FUNCTION_BLOCK "DEVTYPE_ODH_Area"
{ S7_Optimized_Access := 'TRUE' }
VERSION : 1.0
   VAR_INPUT
      "Alarm" { S7_HMI_Accessible := 'False'; S7_HMI_Visible := 'False'} : BOOL;   //EPICS Status variable: Alarm
      "WarmUp" { S7_HMI_Accessible := 'False'; S7_HMI_Visible := 'False'} : BOOL;   //EPICS Status variable: WarmUp
      "ConnLost" { S7_HMI_Accessible := 'False'; S7_HMI_Visible := 'False'} : BOOL;   //EPICS Status variable: ConnLost
   END_VAR
   VAR_OUTPUT
      DEVICE_PARAM_OK { S7_HMI_Accessible := 'False'; S7_HMI_Visible := 'False'} : Bool;
   END_VAR
   VAR_IN_OUT
   END_VAR
   VAR
      StatusReg { S7_HMI_Accessible := 'False'; S7_HMI_Visible := 'False'} : Array[0..0] of Word;
      CommandReg { S7_HMI_Accessible := 'False'; S7_HMI_Visible := 'False'} : Array[0..0] of Word;
   END_VAR
   Var DB_SPECIFIC
      MyWord { S7_HMI_Accessible := 'False'; S7_HMI_Visible := 'False'} : Word;
      MyBytesinWord { S7_HMI_Accessible := 'False'; S7_HMI_Visible := 'False'} AT MyWord : Array[0..1] of Byte;
      MyBoolsinWord { S7_HMI_Accessible := 'False'; S7_HMI_Visible := 'False'} AT MyWord : Array[0..15] of Bool;
      MyDInt { S7_HMI_Accessible := 'False'; S7_HMI_Visible := 'False'} : DInt;
      MyWordsinDint { S7_HMI_Accessible := 'False'; S7_HMI_Visible := 'False'} AT MyDInt : Array[0..1] of Word;
      MyReal { S7_HMI_Accessible := 'False'; S7_HMI_Visible := 'False'} : Real;
      MyWordsinReal { S7_HMI_Accessible := 'False'; S7_HMI_Visible := 'False'} AT MyReal : Array[0..1] of Word;
      MyInt { S7_HMI_Accessible := 'False'; S7_HMI_Visible := 'False'} : Int;
      MyWordinInt { S7_HMI_Accessible := 'False'; S7_HMI_Visible := 'False'} AT MyInt : Word;
      MyDWord { S7_HMI_Accessible := 'False'; S7_HMI_Visible := 'False'} : DWord;
      MyWordsinDWord { S7_HMI_Accessible := 'False'; S7_HMI_Visible := 'False'} AT MyDWord : Array[0..1] of Word;
      MyTime { S7_HMI_Accessible := 'False'; S7_HMI_Visible := 'False'} : Time;
      MyWordsinTime { S7_HMI_Accessible := 'False'; S7_HMI_Visible := 'False'} AT MyTime : Array[0..1] of Word;
   END_VAR
   VAR_TEMP
      HashModbus : DInt;
      HashIFA : DInt;
      HashTIAMap : DInt;
   END_VAR
    //Author: Miklos Boros (miklos.boros@esss.se), Copyrigth 2017-2018 by European Spallation Source, Lund
    //This block was generated by PLCFactory, please don't change it MANUALLY!
    //Input File Name: KG-GTA_ODH-PLC-01-template-IFA-20181024185957.ifa
    //According to HASH: 733470530
    //Device type: ODH_Area
    //Generated: 20181024185959
    //Description: This function does the variable mapping for a device. All device-variable will be linked to an interface variable defined in this block.

    //********************************************
    //****************HASH check******************
    //********************************************


    #MyWordsinDint[0] := "EPICSToPLC"."Word"[0];
    #MyWordsinDint[1] := "EPICSToPLC"."Word"[1];
    #HashModbus := #MyDInt; //Hash from EPICS/ModbusTCP

    #HashIFA := 733470530; //Hash from Interface Factory as a constant

    #MyWordsinDint[0] := "PLCToEPICS"."Word"[0];
    #MyWordsinDint[1] := "PLCToEPICS"."Word"[1];
    #HashTIAMap := #MyDInt; //Hash from PLCFactory TIA Map


    IF ((#HashIFA = #HashModbus) AND (#HashModbus = #HashTIAMap)) THEN //Check CRCs
        #DEVICE_PARAM_OK := TRUE;
       //########################### ODH Detection System   ##############################
       //###########################
       //STATUS BLOCK
       //###########################

    //********************************************
    //*************STATUS VARIABLES***************
    //********************************************


       #MyWord := W#0;
       #MyBoolsinWord[8] := #"Alarm";    //EPICSName: Alarm
       #MyBoolsinWord[9] := #"WarmUp";    //EPICSName: WarmUp
       #MyBoolsinWord[10] := #"ConnLost";    //EPICSName: ConnLost
       #StatusReg[0] := #MyWord;
    Else
       #DEVICE_PARAM_OK := FALSE; //Invalid Hash
    END_IF;
END_FUNCTION_BLOCK
FUNCTION_BLOCK "DEVTYPE_ODH_O2iM"
{ S7_Optimized_Access := 'TRUE' }
VERSION : 1.0
   VAR_INPUT
      "O2Level" { S7_HMI_Accessible := 'False'; S7_HMI_Visible := 'False'} : REAL;   //EPICS Status variable: O2Level
      "ODHAlarm" { S7_HMI_Accessible := 'False'; S7_HMI_Visible := 'False'} : BOOL;   //EPICS Status variable: ODHAlarm
      "ODHWarning" { S7_HMI_Accessible := 'False'; S7_HMI_Visible := 'False'} : BOOL;   //EPICS Status variable: ODHWarning
      "MonitHealthy" { S7_HMI_Accessible := 'False'; S7_HMI_Visible := 'False'} : BOOL;   //EPICS Status variable: MonitHealthy
      "Maint" { S7_HMI_Accessible := 'False'; S7_HMI_Visible := 'False'} : BOOL;   //EPICS Status variable: Maint
      "MonitWarning" { S7_HMI_Accessible := 'False'; S7_HMI_Visible := 'False'} : BOOL;   //EPICS Status variable: MonitWarning
      "SysOK" { S7_HMI_Accessible := 'False'; S7_HMI_Visible := 'False'} : BOOL;   //EPICS Status variable: SysOK
      "WarmUp" { S7_HMI_Accessible := 'False'; S7_HMI_Visible := 'False'} : BOOL;   //EPICS Status variable: WarmUp
      "ConnLost" { S7_HMI_Accessible := 'False'; S7_HMI_Visible := 'False'} : BOOL;   //EPICS Status variable: ConnLost
   END_VAR
   VAR_OUTPUT
      DEVICE_PARAM_OK { S7_HMI_Accessible := 'False'; S7_HMI_Visible := 'False'} : Bool;
   END_VAR
   VAR_IN_OUT
   END_VAR
   VAR
      StatusReg { S7_HMI_Accessible := 'False'; S7_HMI_Visible := 'False'} : Array[0..2] of Word;
      CommandReg { S7_HMI_Accessible := 'False'; S7_HMI_Visible := 'False'} : Array[0..0] of Word;
   END_VAR
   Var DB_SPECIFIC
      MyWord { S7_HMI_Accessible := 'False'; S7_HMI_Visible := 'False'} : Word;
      MyBytesinWord { S7_HMI_Accessible := 'False'; S7_HMI_Visible := 'False'} AT MyWord : Array[0..1] of Byte;
      MyBoolsinWord { S7_HMI_Accessible := 'False'; S7_HMI_Visible := 'False'} AT MyWord : Array[0..15] of Bool;
      MyDInt { S7_HMI_Accessible := 'False'; S7_HMI_Visible := 'False'} : DInt;
      MyWordsinDint { S7_HMI_Accessible := 'False'; S7_HMI_Visible := 'False'} AT MyDInt : Array[0..1] of Word;
      MyReal { S7_HMI_Accessible := 'False'; S7_HMI_Visible := 'False'} : Real;
      MyWordsinReal { S7_HMI_Accessible := 'False'; S7_HMI_Visible := 'False'} AT MyReal : Array[0..1] of Word;
      MyInt { S7_HMI_Accessible := 'False'; S7_HMI_Visible := 'False'} : Int;
      MyWordinInt { S7_HMI_Accessible := 'False'; S7_HMI_Visible := 'False'} AT MyInt : Word;
      MyDWord { S7_HMI_Accessible := 'False'; S7_HMI_Visible := 'False'} : DWord;
      MyWordsinDWord { S7_HMI_Accessible := 'False'; S7_HMI_Visible := 'False'} AT MyDWord : Array[0..1] of Word;
      MyTime { S7_HMI_Accessible := 'False'; S7_HMI_Visible := 'False'} : Time;
      MyWordsinTime { S7_HMI_Accessible := 'False'; S7_HMI_Visible := 'False'} AT MyTime : Array[0..1] of Word;
   END_VAR
   VAR_TEMP
      HashModbus : DInt;
      HashIFA : DInt;
      HashTIAMap : DInt;
   END_VAR
    //Author: Miklos Boros (miklos.boros@esss.se), Copyrigth 2017-2018 by European Spallation Source, Lund
    //This block was generated by PLCFactory, please don't change it MANUALLY!
    //Input File Name: KG-GTA_ODH-PLC-01-template-IFA-20181024185957.ifa
    //According to HASH: 733470530
    //Device type: ODH_O2iM
    //Generated: 20181024185959
    //Description: This function does the variable mapping for a device. All device-variable will be linked to an interface variable defined in this block.

    //********************************************
    //****************HASH check******************
    //********************************************


    #MyWordsinDint[0] := "EPICSToPLC"."Word"[0];
    #MyWordsinDint[1] := "EPICSToPLC"."Word"[1];
    #HashModbus := #MyDInt; //Hash from EPICS/ModbusTCP

    #HashIFA := 733470530; //Hash from Interface Factory as a constant

    #MyWordsinDint[0] := "PLCToEPICS"."Word"[0];
    #MyWordsinDint[1] := "PLCToEPICS"."Word"[1];
    #HashTIAMap := #MyDInt; //Hash from PLCFactory TIA Map


    IF ((#HashIFA = #HashModbus) AND (#HashModbus = #HashTIAMap)) THEN //Check CRCs
        #DEVICE_PARAM_OK := TRUE;
       //########################### ODH Detection System   ##############################
       //###########################
       //STATUS BLOCK
       //###########################

    //********************************************
    //*************STATUS VARIABLES***************
    //********************************************


       #MyReal := #"O2Level";
       #StatusReg[0] := #MyWordsinReal[0];
       #StatusReg[1] := #MyWordsinReal[1];

       #MyWord := W#0;
       #MyBoolsinWord[8] := #"ODHAlarm";    //EPICSName: ODHAlarm
       #MyBoolsinWord[9] := #"ODHWarning";    //EPICSName: ODHWarning
       #MyBoolsinWord[10] := #"MonitHealthy";    //EPICSName: MonitHealthy
       #MyBoolsinWord[11] := #"Maint";    //EPICSName: Maint
       #MyBoolsinWord[12] := #"MonitWarning";    //EPICSName: MonitWarning
       #MyBoolsinWord[13] := #"SysOK";    //EPICSName: SysOK
       #MyBoolsinWord[14] := #"WarmUp";    //EPICSName: WarmUp
       #MyBoolsinWord[15] := #"ConnLost";    //EPICSName: ConnLost
       #StatusReg[2] := #MyWord;
    Else
       #DEVICE_PARAM_OK := FALSE; //Invalid Hash
    END_IF;
END_FUNCTION_BLOCK
FUNCTION_BLOCK "DEVTYPE_ODH_Rack"
{ S7_Optimized_Access := 'TRUE' }
VERSION : 1.0
   VAR_INPUT
      "SurgeArrOK" { S7_HMI_Accessible := 'False'; S7_HMI_Visible := 'False'} : BOOL;   //EPICS Status variable: SurgeArrOK
      "PS24vOK" { S7_HMI_Accessible := 'False'; S7_HMI_Visible := 'False'} : BOOL;   //EPICS Status variable: PS24vOK
      "UPSBatOK" { S7_HMI_Accessible := 'False'; S7_HMI_Visible := 'False'} : BOOL;   //EPICS Status variable: UPSBatOK
      "UPS24vOK" { S7_HMI_Accessible := 'False'; S7_HMI_Visible := 'False'} : BOOL;   //EPICS Status variable: UPS24vOK
      "UPSBuffReady" { S7_HMI_Accessible := 'False'; S7_HMI_Visible := 'False'} : BOOL;   //EPICS Status variable: UPSBuffReady
      "UPSBatt85" { S7_HMI_Accessible := 'False'; S7_HMI_Visible := 'False'} : BOOL;   //EPICS Status variable: UPSBatt85
      "UPSAlarm" { S7_HMI_Accessible := 'False'; S7_HMI_Visible := 'False'} : BOOL;   //EPICS Status variable: UPSAlarm
   END_VAR
   VAR_OUTPUT
      DEVICE_PARAM_OK { S7_HMI_Accessible := 'False'; S7_HMI_Visible := 'False'} : Bool;
   END_VAR
   VAR_IN_OUT
   END_VAR
   VAR
      StatusReg { S7_HMI_Accessible := 'False'; S7_HMI_Visible := 'False'} : Array[0..0] of Word;
      CommandReg { S7_HMI_Accessible := 'False'; S7_HMI_Visible := 'False'} : Array[0..0] of Word;
   END_VAR
   Var DB_SPECIFIC
      MyWord { S7_HMI_Accessible := 'False'; S7_HMI_Visible := 'False'} : Word;
      MyBytesinWord { S7_HMI_Accessible := 'False'; S7_HMI_Visible := 'False'} AT MyWord : Array[0..1] of Byte;
      MyBoolsinWord { S7_HMI_Accessible := 'False'; S7_HMI_Visible := 'False'} AT MyWord : Array[0..15] of Bool;
      MyDInt { S7_HMI_Accessible := 'False'; S7_HMI_Visible := 'False'} : DInt;
      MyWordsinDint { S7_HMI_Accessible := 'False'; S7_HMI_Visible := 'False'} AT MyDInt : Array[0..1] of Word;
      MyReal { S7_HMI_Accessible := 'False'; S7_HMI_Visible := 'False'} : Real;
      MyWordsinReal { S7_HMI_Accessible := 'False'; S7_HMI_Visible := 'False'} AT MyReal : Array[0..1] of Word;
      MyInt { S7_HMI_Accessible := 'False'; S7_HMI_Visible := 'False'} : Int;
      MyWordinInt { S7_HMI_Accessible := 'False'; S7_HMI_Visible := 'False'} AT MyInt : Word;
      MyDWord { S7_HMI_Accessible := 'False'; S7_HMI_Visible := 'False'} : DWord;
      MyWordsinDWord { S7_HMI_Accessible := 'False'; S7_HMI_Visible := 'False'} AT MyDWord : Array[0..1] of Word;
      MyTime { S7_HMI_Accessible := 'False'; S7_HMI_Visible := 'False'} : Time;
      MyWordsinTime { S7_HMI_Accessible := 'False'; S7_HMI_Visible := 'False'} AT MyTime : Array[0..1] of Word;
   END_VAR
   VAR_TEMP
      HashModbus : DInt;
      HashIFA : DInt;
      HashTIAMap : DInt;
   END_VAR
    //Author: Miklos Boros (miklos.boros@esss.se), Copyrigth 2017-2018 by European Spallation Source, Lund
    //This block was generated by PLCFactory, please don't change it MANUALLY!
    //Input File Name: KG-GTA_ODH-PLC-01-template-IFA-20181024185957.ifa
    //According to HASH: 733470530
    //Device type: ODH_Rack
    //Generated: 20181024185959
    //Description: This function does the variable mapping for a device. All device-variable will be linked to an interface variable defined in this block.

    //********************************************
    //****************HASH check******************
    //********************************************


    #MyWordsinDint[0] := "EPICSToPLC"."Word"[0];
    #MyWordsinDint[1] := "EPICSToPLC"."Word"[1];
    #HashModbus := #MyDInt; //Hash from EPICS/ModbusTCP

    #HashIFA := 733470530; //Hash from Interface Factory as a constant

    #MyWordsinDint[0] := "PLCToEPICS"."Word"[0];
    #MyWordsinDint[1] := "PLCToEPICS"."Word"[1];
    #HashTIAMap := #MyDInt; //Hash from PLCFactory TIA Map


    IF ((#HashIFA = #HashModbus) AND (#HashModbus = #HashTIAMap)) THEN //Check CRCs
        #DEVICE_PARAM_OK := TRUE;
       //########################### ODH Detection System   ##############################
       //###########################
       //STATUS BLOCK
       //###########################

    //********************************************
    //*************STATUS VARIABLES***************
    //********************************************


       #MyWord := W#0;
       #MyBoolsinWord[8] := #"SurgeArrOK";    //EPICSName: SurgeArrOK
       #MyBoolsinWord[9] := #"PS24vOK";    //EPICSName: PS24vOK
       #MyBoolsinWord[10] := #"UPSBatOK";    //EPICSName: UPSBatOK
       #MyBoolsinWord[11] := #"UPS24vOK";    //EPICSName: UPS24vOK
       #MyBoolsinWord[12] := #"UPSBuffReady";    //EPICSName: UPSBuffReady
       #MyBoolsinWord[13] := #"UPSBatt85";    //EPICSName: UPSBatt85
       #MyBoolsinWord[14] := #"UPSAlarm";    //EPICSName: UPSAlarm
       #StatusReg[0] := #MyWord;
    Else
       #DEVICE_PARAM_OK := FALSE; //Invalid Hash
    END_IF;
END_FUNCTION_BLOCK

DATA_BLOCK "DEV_CTLG-CS:ODH-Area_iDB"
{ S7_Optimized_Access := 'TRUE' }
VERSION : 1.0
NON_RETAIN
"DEVTYPE_ODH_Area"
BEGIN
END_DATA_BLOCK


DATA_BLOCK "DEV_CXB-CXH:ODH-Area_iDB"
{ S7_Optimized_Access := 'TRUE' }
VERSION : 1.0
NON_RETAIN
"DEVTYPE_ODH_Area"
BEGIN
END_DATA_BLOCK


DATA_BLOCK "DEV_CTLG-CS:ODH-O2iM-20_iDB"
{ S7_Optimized_Access := 'TRUE' }
VERSION : 1.0
NON_RETAIN
"DEVTYPE_ODH_O2iM"
BEGIN
END_DATA_BLOCK


DATA_BLOCK "DEV_CTLG-CS:ODH-O2iM-21_iDB"
{ S7_Optimized_Access := 'TRUE' }
VERSION : 1.0
NON_RETAIN
"DEVTYPE_ODH_O2iM"
BEGIN
END_DATA_BLOCK


DATA_BLOCK "DEV_CTLG-CS:ODH-O2iM-22_iDB"
{ S7_Optimized_Access := 'TRUE' }
VERSION : 1.0
NON_RETAIN
"DEVTYPE_ODH_O2iM"
BEGIN
END_DATA_BLOCK


DATA_BLOCK "DEV_CXB-CXH:ODH-O2iM-13_iDB"
{ S7_Optimized_Access := 'TRUE' }
VERSION : 1.0
NON_RETAIN
"DEVTYPE_ODH_O2iM"
BEGIN
END_DATA_BLOCK


DATA_BLOCK "DEV_CXB-CXH:ODH-O2iM-14_iDB"
{ S7_Optimized_Access := 'TRUE' }
VERSION : 1.0
NON_RETAIN
"DEVTYPE_ODH_O2iM"
BEGIN
END_DATA_BLOCK


DATA_BLOCK "DEV_CXB-CXH:ODH-O2iM-15_iDB"
{ S7_Optimized_Access := 'TRUE' }
VERSION : 1.0
NON_RETAIN
"DEVTYPE_ODH_O2iM"
BEGIN
END_DATA_BLOCK


DATA_BLOCK "DEV_CXB-CXH:ODH-O2iM-16_iDB"
{ S7_Optimized_Access := 'TRUE' }
VERSION : 1.0
NON_RETAIN
"DEVTYPE_ODH_O2iM"
BEGIN
END_DATA_BLOCK


DATA_BLOCK "DEV_CXB-CXH:ODH-O2iM-17_iDB"
{ S7_Optimized_Access := 'TRUE' }
VERSION : 1.0
NON_RETAIN
"DEVTYPE_ODH_O2iM"
BEGIN
END_DATA_BLOCK


DATA_BLOCK "DEV_CXB-CXH:ODH-O2iM-18_iDB"
{ S7_Optimized_Access := 'TRUE' }
VERSION : 1.0
NON_RETAIN
"DEVTYPE_ODH_O2iM"
BEGIN
END_DATA_BLOCK


DATA_BLOCK "DEV_CXB-CXH:ODH-O2iM-19_iDB"
{ S7_Optimized_Access := 'TRUE' }
VERSION : 1.0
NON_RETAIN
"DEVTYPE_ODH_O2iM"
BEGIN
END_DATA_BLOCK


DATA_BLOCK "DEV_HCB-ACH:ODH-O2iM-1_iDB"
{ S7_Optimized_Access := 'TRUE' }
VERSION : 1.0
NON_RETAIN
"DEVTYPE_ODH_O2iM"
BEGIN
END_DATA_BLOCK


DATA_BLOCK "DEV_HCB-ACH:ODH-O2iM-2_iDB"
{ S7_Optimized_Access := 'TRUE' }
VERSION : 1.0
NON_RETAIN
"DEVTYPE_ODH_O2iM"
BEGIN
END_DATA_BLOCK


DATA_BLOCK "DEV_HCB-ACH:ODH-O2iM-3_iDB"
{ S7_Optimized_Access := 'TRUE' }
VERSION : 1.0
NON_RETAIN
"DEVTYPE_ODH_O2iM"
BEGIN
END_DATA_BLOCK


DATA_BLOCK "DEV_HCB-ACH:ODH-O2iM-4_iDB"
{ S7_Optimized_Access := 'TRUE' }
VERSION : 1.0
NON_RETAIN
"DEVTYPE_ODH_O2iM"
BEGIN
END_DATA_BLOCK


DATA_BLOCK "DEV_HCB-ACH:ODH-O2iM-5_iDB"
{ S7_Optimized_Access := 'TRUE' }
VERSION : 1.0
NON_RETAIN
"DEVTYPE_ODH_O2iM"
BEGIN
END_DATA_BLOCK


DATA_BLOCK "DEV_HCB-DogSh:ODH-O2iM-12_iDB"
{ S7_Optimized_Access := 'TRUE' }
VERSION : 1.0
NON_RETAIN
"DEVTYPE_ODH_O2iM"
BEGIN
END_DATA_BLOCK


DATA_BLOCK "DEV_HCB-HPGS:ODH-O2iM-10_iDB"
{ S7_Optimized_Access := 'TRUE' }
VERSION : 1.0
NON_RETAIN
"DEVTYPE_ODH_O2iM"
BEGIN
END_DATA_BLOCK


DATA_BLOCK "DEV_HCB-HPGS:ODH-O2iM-11_iDB"
{ S7_Optimized_Access := 'TRUE' }
VERSION : 1.0
NON_RETAIN
"DEVTYPE_ODH_O2iM"
BEGIN
END_DATA_BLOCK


DATA_BLOCK "DEV_HCB-TCH:ODH-O2iM-6_iDB"
{ S7_Optimized_Access := 'TRUE' }
VERSION : 1.0
NON_RETAIN
"DEVTYPE_ODH_O2iM"
BEGIN
END_DATA_BLOCK


DATA_BLOCK "DEV_HCB-TCH:ODH-O2iM-7_iDB"
{ S7_Optimized_Access := 'TRUE' }
VERSION : 1.0
NON_RETAIN
"DEVTYPE_ODH_O2iM"
BEGIN
END_DATA_BLOCK


DATA_BLOCK "DEV_HCB-TCH:ODH-O2iM-8_iDB"
{ S7_Optimized_Access := 'TRUE' }
VERSION : 1.0
NON_RETAIN
"DEVTYPE_ODH_O2iM"
BEGIN
END_DATA_BLOCK


DATA_BLOCK "DEV_HCB-TCH:ODH-O2iM-9_iDB"
{ S7_Optimized_Access := 'TRUE' }
VERSION : 1.0
NON_RETAIN
"DEVTYPE_ODH_O2iM"
BEGIN
END_DATA_BLOCK


DATA_BLOCK "DEV_CXB-CXH:ODH-RIO-2_iDB"
{ S7_Optimized_Access := 'TRUE' }
VERSION : 1.0
NON_RETAIN
"DEVTYPE_ODH_Rack"
BEGIN
END_DATA_BLOCK


DATA_BLOCK "DEV_HCB-ACH:ODH-RIO-1_iDB"
{ S7_Optimized_Access := 'TRUE' }
VERSION : 1.0
NON_RETAIN
"DEVTYPE_ODH_Rack"
BEGIN
END_DATA_BLOCK


DATA_BLOCK "DEV_TS2-020Row:CnPw-U-001_iDB"
{ S7_Optimized_Access := 'TRUE' }
VERSION : 1.0
NON_RETAIN
"DEVTYPE_ODH_Rack"
BEGIN
END_DATA_BLOCK

DATA_BLOCK "EPICS_PLC_Tester"
{ S7_Optimized_Access := 'FALSE' }
VERSION : 0.1
NON_RETAIN
   STRUCT
      HeartBeat { S7_HMI_Accessible := 'False'; S7_HMI_Visible := 'False'} : Bool;
      "CTLG-CS:ODH-Area_Alarm" { S7_HMI_Accessible := 'False'; S7_HMI_Visible := 'False'} : BOOL;   //EPICS Status variable: Alarm
      "CTLG-CS:ODH-Area_WarmUp" { S7_HMI_Accessible := 'False'; S7_HMI_Visible := 'False'} : BOOL;   //EPICS Status variable: WarmUp
      "CTLG-CS:ODH-Area_ConnLost" { S7_HMI_Accessible := 'False'; S7_HMI_Visible := 'False'} : BOOL;   //EPICS Status variable: ConnLost
      "CXB-CXH:ODH-Area_Alarm" { S7_HMI_Accessible := 'False'; S7_HMI_Visible := 'False'} : BOOL;   //EPICS Status variable: Alarm
      "CXB-CXH:ODH-Area_WarmUp" { S7_HMI_Accessible := 'False'; S7_HMI_Visible := 'False'} : BOOL;   //EPICS Status variable: WarmUp
      "CXB-CXH:ODH-Area_ConnLost" { S7_HMI_Accessible := 'False'; S7_HMI_Visible := 'False'} : BOOL;   //EPICS Status variable: ConnLost
      "CTLG-CS:ODH-O2iM-20_O2Level" { S7_HMI_Accessible := 'False'; S7_HMI_Visible := 'False'} : REAL;   //EPICS Status variable: O2Level
      "CTLG-CS:ODH-O2iM-20_ODHAlarm" { S7_HMI_Accessible := 'False'; S7_HMI_Visible := 'False'} : BOOL;   //EPICS Status variable: ODHAlarm
      "CTLG-CS:ODH-O2iM-20_ODHWarning" { S7_HMI_Accessible := 'False'; S7_HMI_Visible := 'False'} : BOOL;   //EPICS Status variable: ODHWarning
      "CTLG-CS:ODH-O2iM-20_MonitHealthy" { S7_HMI_Accessible := 'False'; S7_HMI_Visible := 'False'} : BOOL;   //EPICS Status variable: MonitHealthy
      "CTLG-CS:ODH-O2iM-20_Maint" { S7_HMI_Accessible := 'False'; S7_HMI_Visible := 'False'} : BOOL;   //EPICS Status variable: Maint
      "CTLG-CS:ODH-O2iM-20_MonitWarning" { S7_HMI_Accessible := 'False'; S7_HMI_Visible := 'False'} : BOOL;   //EPICS Status variable: MonitWarning
      "CTLG-CS:ODH-O2iM-20_SysOK" { S7_HMI_Accessible := 'False'; S7_HMI_Visible := 'False'} : BOOL;   //EPICS Status variable: SysOK
      "CTLG-CS:ODH-O2iM-20_WarmUp" { S7_HMI_Accessible := 'False'; S7_HMI_Visible := 'False'} : BOOL;   //EPICS Status variable: WarmUp
      "CTLG-CS:ODH-O2iM-20_ConnLost" { S7_HMI_Accessible := 'False'; S7_HMI_Visible := 'False'} : BOOL;   //EPICS Status variable: ConnLost
      "CTLG-CS:ODH-O2iM-21_O2Level" { S7_HMI_Accessible := 'False'; S7_HMI_Visible := 'False'} : REAL;   //EPICS Status variable: O2Level
      "CTLG-CS:ODH-O2iM-21_ODHAlarm" { S7_HMI_Accessible := 'False'; S7_HMI_Visible := 'False'} : BOOL;   //EPICS Status variable: ODHAlarm
      "CTLG-CS:ODH-O2iM-21_ODHWarning" { S7_HMI_Accessible := 'False'; S7_HMI_Visible := 'False'} : BOOL;   //EPICS Status variable: ODHWarning
      "CTLG-CS:ODH-O2iM-21_MonitHealthy" { S7_HMI_Accessible := 'False'; S7_HMI_Visible := 'False'} : BOOL;   //EPICS Status variable: MonitHealthy
      "CTLG-CS:ODH-O2iM-21_Maint" { S7_HMI_Accessible := 'False'; S7_HMI_Visible := 'False'} : BOOL;   //EPICS Status variable: Maint
      "CTLG-CS:ODH-O2iM-21_MonitWarning" { S7_HMI_Accessible := 'False'; S7_HMI_Visible := 'False'} : BOOL;   //EPICS Status variable: MonitWarning
      "CTLG-CS:ODH-O2iM-21_SysOK" { S7_HMI_Accessible := 'False'; S7_HMI_Visible := 'False'} : BOOL;   //EPICS Status variable: SysOK
      "CTLG-CS:ODH-O2iM-21_WarmUp" { S7_HMI_Accessible := 'False'; S7_HMI_Visible := 'False'} : BOOL;   //EPICS Status variable: WarmUp
      "CTLG-CS:ODH-O2iM-21_ConnLost" { S7_HMI_Accessible := 'False'; S7_HMI_Visible := 'False'} : BOOL;   //EPICS Status variable: ConnLost
      "CTLG-CS:ODH-O2iM-22_O2Level" { S7_HMI_Accessible := 'False'; S7_HMI_Visible := 'False'} : REAL;   //EPICS Status variable: O2Level
      "CTLG-CS:ODH-O2iM-22_ODHAlarm" { S7_HMI_Accessible := 'False'; S7_HMI_Visible := 'False'} : BOOL;   //EPICS Status variable: ODHAlarm
      "CTLG-CS:ODH-O2iM-22_ODHWarning" { S7_HMI_Accessible := 'False'; S7_HMI_Visible := 'False'} : BOOL;   //EPICS Status variable: ODHWarning
      "CTLG-CS:ODH-O2iM-22_MonitHealthy" { S7_HMI_Accessible := 'False'; S7_HMI_Visible := 'False'} : BOOL;   //EPICS Status variable: MonitHealthy
      "CTLG-CS:ODH-O2iM-22_Maint" { S7_HMI_Accessible := 'False'; S7_HMI_Visible := 'False'} : BOOL;   //EPICS Status variable: Maint
      "CTLG-CS:ODH-O2iM-22_MonitWarning" { S7_HMI_Accessible := 'False'; S7_HMI_Visible := 'False'} : BOOL;   //EPICS Status variable: MonitWarning
      "CTLG-CS:ODH-O2iM-22_SysOK" { S7_HMI_Accessible := 'False'; S7_HMI_Visible := 'False'} : BOOL;   //EPICS Status variable: SysOK
      "CTLG-CS:ODH-O2iM-22_WarmUp" { S7_HMI_Accessible := 'False'; S7_HMI_Visible := 'False'} : BOOL;   //EPICS Status variable: WarmUp
      "CTLG-CS:ODH-O2iM-22_ConnLost" { S7_HMI_Accessible := 'False'; S7_HMI_Visible := 'False'} : BOOL;   //EPICS Status variable: ConnLost
      "CXB-CXH:ODH-O2iM-13_O2Level" { S7_HMI_Accessible := 'False'; S7_HMI_Visible := 'False'} : REAL;   //EPICS Status variable: O2Level
      "CXB-CXH:ODH-O2iM-13_ODHAlarm" { S7_HMI_Accessible := 'False'; S7_HMI_Visible := 'False'} : BOOL;   //EPICS Status variable: ODHAlarm
      "CXB-CXH:ODH-O2iM-13_ODHWarning" { S7_HMI_Accessible := 'False'; S7_HMI_Visible := 'False'} : BOOL;   //EPICS Status variable: ODHWarning
      "CXB-CXH:ODH-O2iM-13_MonitHealthy" { S7_HMI_Accessible := 'False'; S7_HMI_Visible := 'False'} : BOOL;   //EPICS Status variable: MonitHealthy
      "CXB-CXH:ODH-O2iM-13_Maint" { S7_HMI_Accessible := 'False'; S7_HMI_Visible := 'False'} : BOOL;   //EPICS Status variable: Maint
      "CXB-CXH:ODH-O2iM-13_MonitWarning" { S7_HMI_Accessible := 'False'; S7_HMI_Visible := 'False'} : BOOL;   //EPICS Status variable: MonitWarning
      "CXB-CXH:ODH-O2iM-13_SysOK" { S7_HMI_Accessible := 'False'; S7_HMI_Visible := 'False'} : BOOL;   //EPICS Status variable: SysOK
      "CXB-CXH:ODH-O2iM-13_WarmUp" { S7_HMI_Accessible := 'False'; S7_HMI_Visible := 'False'} : BOOL;   //EPICS Status variable: WarmUp
      "CXB-CXH:ODH-O2iM-13_ConnLost" { S7_HMI_Accessible := 'False'; S7_HMI_Visible := 'False'} : BOOL;   //EPICS Status variable: ConnLost
      "CXB-CXH:ODH-O2iM-14_O2Level" { S7_HMI_Accessible := 'False'; S7_HMI_Visible := 'False'} : REAL;   //EPICS Status variable: O2Level
      "CXB-CXH:ODH-O2iM-14_ODHAlarm" { S7_HMI_Accessible := 'False'; S7_HMI_Visible := 'False'} : BOOL;   //EPICS Status variable: ODHAlarm
      "CXB-CXH:ODH-O2iM-14_ODHWarning" { S7_HMI_Accessible := 'False'; S7_HMI_Visible := 'False'} : BOOL;   //EPICS Status variable: ODHWarning
      "CXB-CXH:ODH-O2iM-14_MonitHealthy" { S7_HMI_Accessible := 'False'; S7_HMI_Visible := 'False'} : BOOL;   //EPICS Status variable: MonitHealthy
      "CXB-CXH:ODH-O2iM-14_Maint" { S7_HMI_Accessible := 'False'; S7_HMI_Visible := 'False'} : BOOL;   //EPICS Status variable: Maint
      "CXB-CXH:ODH-O2iM-14_MonitWarning" { S7_HMI_Accessible := 'False'; S7_HMI_Visible := 'False'} : BOOL;   //EPICS Status variable: MonitWarning
      "CXB-CXH:ODH-O2iM-14_SysOK" { S7_HMI_Accessible := 'False'; S7_HMI_Visible := 'False'} : BOOL;   //EPICS Status variable: SysOK
      "CXB-CXH:ODH-O2iM-14_WarmUp" { S7_HMI_Accessible := 'False'; S7_HMI_Visible := 'False'} : BOOL;   //EPICS Status variable: WarmUp
      "CXB-CXH:ODH-O2iM-14_ConnLost" { S7_HMI_Accessible := 'False'; S7_HMI_Visible := 'False'} : BOOL;   //EPICS Status variable: ConnLost
      "CXB-CXH:ODH-O2iM-15_O2Level" { S7_HMI_Accessible := 'False'; S7_HMI_Visible := 'False'} : REAL;   //EPICS Status variable: O2Level
      "CXB-CXH:ODH-O2iM-15_ODHAlarm" { S7_HMI_Accessible := 'False'; S7_HMI_Visible := 'False'} : BOOL;   //EPICS Status variable: ODHAlarm
      "CXB-CXH:ODH-O2iM-15_ODHWarning" { S7_HMI_Accessible := 'False'; S7_HMI_Visible := 'False'} : BOOL;   //EPICS Status variable: ODHWarning
      "CXB-CXH:ODH-O2iM-15_MonitHealthy" { S7_HMI_Accessible := 'False'; S7_HMI_Visible := 'False'} : BOOL;   //EPICS Status variable: MonitHealthy
      "CXB-CXH:ODH-O2iM-15_Maint" { S7_HMI_Accessible := 'False'; S7_HMI_Visible := 'False'} : BOOL;   //EPICS Status variable: Maint
      "CXB-CXH:ODH-O2iM-15_MonitWarning" { S7_HMI_Accessible := 'False'; S7_HMI_Visible := 'False'} : BOOL;   //EPICS Status variable: MonitWarning
      "CXB-CXH:ODH-O2iM-15_SysOK" { S7_HMI_Accessible := 'False'; S7_HMI_Visible := 'False'} : BOOL;   //EPICS Status variable: SysOK
      "CXB-CXH:ODH-O2iM-15_WarmUp" { S7_HMI_Accessible := 'False'; S7_HMI_Visible := 'False'} : BOOL;   //EPICS Status variable: WarmUp
      "CXB-CXH:ODH-O2iM-15_ConnLost" { S7_HMI_Accessible := 'False'; S7_HMI_Visible := 'False'} : BOOL;   //EPICS Status variable: ConnLost
      "CXB-CXH:ODH-O2iM-16_O2Level" { S7_HMI_Accessible := 'False'; S7_HMI_Visible := 'False'} : REAL;   //EPICS Status variable: O2Level
      "CXB-CXH:ODH-O2iM-16_ODHAlarm" { S7_HMI_Accessible := 'False'; S7_HMI_Visible := 'False'} : BOOL;   //EPICS Status variable: ODHAlarm
      "CXB-CXH:ODH-O2iM-16_ODHWarning" { S7_HMI_Accessible := 'False'; S7_HMI_Visible := 'False'} : BOOL;   //EPICS Status variable: ODHWarning
      "CXB-CXH:ODH-O2iM-16_MonitHealthy" { S7_HMI_Accessible := 'False'; S7_HMI_Visible := 'False'} : BOOL;   //EPICS Status variable: MonitHealthy
      "CXB-CXH:ODH-O2iM-16_Maint" { S7_HMI_Accessible := 'False'; S7_HMI_Visible := 'False'} : BOOL;   //EPICS Status variable: Maint
      "CXB-CXH:ODH-O2iM-16_MonitWarning" { S7_HMI_Accessible := 'False'; S7_HMI_Visible := 'False'} : BOOL;   //EPICS Status variable: MonitWarning
      "CXB-CXH:ODH-O2iM-16_SysOK" { S7_HMI_Accessible := 'False'; S7_HMI_Visible := 'False'} : BOOL;   //EPICS Status variable: SysOK
      "CXB-CXH:ODH-O2iM-16_WarmUp" { S7_HMI_Accessible := 'False'; S7_HMI_Visible := 'False'} : BOOL;   //EPICS Status variable: WarmUp
      "CXB-CXH:ODH-O2iM-16_ConnLost" { S7_HMI_Accessible := 'False'; S7_HMI_Visible := 'False'} : BOOL;   //EPICS Status variable: ConnLost
      "CXB-CXH:ODH-O2iM-17_O2Level" { S7_HMI_Accessible := 'False'; S7_HMI_Visible := 'False'} : REAL;   //EPICS Status variable: O2Level
      "CXB-CXH:ODH-O2iM-17_ODHAlarm" { S7_HMI_Accessible := 'False'; S7_HMI_Visible := 'False'} : BOOL;   //EPICS Status variable: ODHAlarm
      "CXB-CXH:ODH-O2iM-17_ODHWarning" { S7_HMI_Accessible := 'False'; S7_HMI_Visible := 'False'} : BOOL;   //EPICS Status variable: ODHWarning
      "CXB-CXH:ODH-O2iM-17_MonitHealthy" { S7_HMI_Accessible := 'False'; S7_HMI_Visible := 'False'} : BOOL;   //EPICS Status variable: MonitHealthy
      "CXB-CXH:ODH-O2iM-17_Maint" { S7_HMI_Accessible := 'False'; S7_HMI_Visible := 'False'} : BOOL;   //EPICS Status variable: Maint
      "CXB-CXH:ODH-O2iM-17_MonitWarning" { S7_HMI_Accessible := 'False'; S7_HMI_Visible := 'False'} : BOOL;   //EPICS Status variable: MonitWarning
      "CXB-CXH:ODH-O2iM-17_SysOK" { S7_HMI_Accessible := 'False'; S7_HMI_Visible := 'False'} : BOOL;   //EPICS Status variable: SysOK
      "CXB-CXH:ODH-O2iM-17_WarmUp" { S7_HMI_Accessible := 'False'; S7_HMI_Visible := 'False'} : BOOL;   //EPICS Status variable: WarmUp
      "CXB-CXH:ODH-O2iM-17_ConnLost" { S7_HMI_Accessible := 'False'; S7_HMI_Visible := 'False'} : BOOL;   //EPICS Status variable: ConnLost
      "CXB-CXH:ODH-O2iM-18_O2Level" { S7_HMI_Accessible := 'False'; S7_HMI_Visible := 'False'} : REAL;   //EPICS Status variable: O2Level
      "CXB-CXH:ODH-O2iM-18_ODHAlarm" { S7_HMI_Accessible := 'False'; S7_HMI_Visible := 'False'} : BOOL;   //EPICS Status variable: ODHAlarm
      "CXB-CXH:ODH-O2iM-18_ODHWarning" { S7_HMI_Accessible := 'False'; S7_HMI_Visible := 'False'} : BOOL;   //EPICS Status variable: ODHWarning
      "CXB-CXH:ODH-O2iM-18_MonitHealthy" { S7_HMI_Accessible := 'False'; S7_HMI_Visible := 'False'} : BOOL;   //EPICS Status variable: MonitHealthy
      "CXB-CXH:ODH-O2iM-18_Maint" { S7_HMI_Accessible := 'False'; S7_HMI_Visible := 'False'} : BOOL;   //EPICS Status variable: Maint
      "CXB-CXH:ODH-O2iM-18_MonitWarning" { S7_HMI_Accessible := 'False'; S7_HMI_Visible := 'False'} : BOOL;   //EPICS Status variable: MonitWarning
      "CXB-CXH:ODH-O2iM-18_SysOK" { S7_HMI_Accessible := 'False'; S7_HMI_Visible := 'False'} : BOOL;   //EPICS Status variable: SysOK
      "CXB-CXH:ODH-O2iM-18_WarmUp" { S7_HMI_Accessible := 'False'; S7_HMI_Visible := 'False'} : BOOL;   //EPICS Status variable: WarmUp
      "CXB-CXH:ODH-O2iM-18_ConnLost" { S7_HMI_Accessible := 'False'; S7_HMI_Visible := 'False'} : BOOL;   //EPICS Status variable: ConnLost
      "CXB-CXH:ODH-O2iM-19_O2Level" { S7_HMI_Accessible := 'False'; S7_HMI_Visible := 'False'} : REAL;   //EPICS Status variable: O2Level
      "CXB-CXH:ODH-O2iM-19_ODHAlarm" { S7_HMI_Accessible := 'False'; S7_HMI_Visible := 'False'} : BOOL;   //EPICS Status variable: ODHAlarm
      "CXB-CXH:ODH-O2iM-19_ODHWarning" { S7_HMI_Accessible := 'False'; S7_HMI_Visible := 'False'} : BOOL;   //EPICS Status variable: ODHWarning
      "CXB-CXH:ODH-O2iM-19_MonitHealthy" { S7_HMI_Accessible := 'False'; S7_HMI_Visible := 'False'} : BOOL;   //EPICS Status variable: MonitHealthy
      "CXB-CXH:ODH-O2iM-19_Maint" { S7_HMI_Accessible := 'False'; S7_HMI_Visible := 'False'} : BOOL;   //EPICS Status variable: Maint
      "CXB-CXH:ODH-O2iM-19_MonitWarning" { S7_HMI_Accessible := 'False'; S7_HMI_Visible := 'False'} : BOOL;   //EPICS Status variable: MonitWarning
      "CXB-CXH:ODH-O2iM-19_SysOK" { S7_HMI_Accessible := 'False'; S7_HMI_Visible := 'False'} : BOOL;   //EPICS Status variable: SysOK
      "CXB-CXH:ODH-O2iM-19_WarmUp" { S7_HMI_Accessible := 'False'; S7_HMI_Visible := 'False'} : BOOL;   //EPICS Status variable: WarmUp
      "CXB-CXH:ODH-O2iM-19_ConnLost" { S7_HMI_Accessible := 'False'; S7_HMI_Visible := 'False'} : BOOL;   //EPICS Status variable: ConnLost
      "HCB-ACH:ODH-O2iM-1_O2Level" { S7_HMI_Accessible := 'False'; S7_HMI_Visible := 'False'} : REAL;   //EPICS Status variable: O2Level
      "HCB-ACH:ODH-O2iM-1_ODHAlarm" { S7_HMI_Accessible := 'False'; S7_HMI_Visible := 'False'} : BOOL;   //EPICS Status variable: ODHAlarm
      "HCB-ACH:ODH-O2iM-1_ODHWarning" { S7_HMI_Accessible := 'False'; S7_HMI_Visible := 'False'} : BOOL;   //EPICS Status variable: ODHWarning
      "HCB-ACH:ODH-O2iM-1_MonitHealthy" { S7_HMI_Accessible := 'False'; S7_HMI_Visible := 'False'} : BOOL;   //EPICS Status variable: MonitHealthy
      "HCB-ACH:ODH-O2iM-1_Maint" { S7_HMI_Accessible := 'False'; S7_HMI_Visible := 'False'} : BOOL;   //EPICS Status variable: Maint
      "HCB-ACH:ODH-O2iM-1_MonitWarning" { S7_HMI_Accessible := 'False'; S7_HMI_Visible := 'False'} : BOOL;   //EPICS Status variable: MonitWarning
      "HCB-ACH:ODH-O2iM-1_SysOK" { S7_HMI_Accessible := 'False'; S7_HMI_Visible := 'False'} : BOOL;   //EPICS Status variable: SysOK
      "HCB-ACH:ODH-O2iM-1_WarmUp" { S7_HMI_Accessible := 'False'; S7_HMI_Visible := 'False'} : BOOL;   //EPICS Status variable: WarmUp
      "HCB-ACH:ODH-O2iM-1_ConnLost" { S7_HMI_Accessible := 'False'; S7_HMI_Visible := 'False'} : BOOL;   //EPICS Status variable: ConnLost
      "HCB-ACH:ODH-O2iM-2_O2Level" { S7_HMI_Accessible := 'False'; S7_HMI_Visible := 'False'} : REAL;   //EPICS Status variable: O2Level
      "HCB-ACH:ODH-O2iM-2_ODHAlarm" { S7_HMI_Accessible := 'False'; S7_HMI_Visible := 'False'} : BOOL;   //EPICS Status variable: ODHAlarm
      "HCB-ACH:ODH-O2iM-2_ODHWarning" { S7_HMI_Accessible := 'False'; S7_HMI_Visible := 'False'} : BOOL;   //EPICS Status variable: ODHWarning
      "HCB-ACH:ODH-O2iM-2_MonitHealthy" { S7_HMI_Accessible := 'False'; S7_HMI_Visible := 'False'} : BOOL;   //EPICS Status variable: MonitHealthy
      "HCB-ACH:ODH-O2iM-2_Maint" { S7_HMI_Accessible := 'False'; S7_HMI_Visible := 'False'} : BOOL;   //EPICS Status variable: Maint
      "HCB-ACH:ODH-O2iM-2_MonitWarning" { S7_HMI_Accessible := 'False'; S7_HMI_Visible := 'False'} : BOOL;   //EPICS Status variable: MonitWarning
      "HCB-ACH:ODH-O2iM-2_SysOK" { S7_HMI_Accessible := 'False'; S7_HMI_Visible := 'False'} : BOOL;   //EPICS Status variable: SysOK
      "HCB-ACH:ODH-O2iM-2_WarmUp" { S7_HMI_Accessible := 'False'; S7_HMI_Visible := 'False'} : BOOL;   //EPICS Status variable: WarmUp
      "HCB-ACH:ODH-O2iM-2_ConnLost" { S7_HMI_Accessible := 'False'; S7_HMI_Visible := 'False'} : BOOL;   //EPICS Status variable: ConnLost
      "HCB-ACH:ODH-O2iM-3_O2Level" { S7_HMI_Accessible := 'False'; S7_HMI_Visible := 'False'} : REAL;   //EPICS Status variable: O2Level
      "HCB-ACH:ODH-O2iM-3_ODHAlarm" { S7_HMI_Accessible := 'False'; S7_HMI_Visible := 'False'} : BOOL;   //EPICS Status variable: ODHAlarm
      "HCB-ACH:ODH-O2iM-3_ODHWarning" { S7_HMI_Accessible := 'False'; S7_HMI_Visible := 'False'} : BOOL;   //EPICS Status variable: ODHWarning
      "HCB-ACH:ODH-O2iM-3_MonitHealthy" { S7_HMI_Accessible := 'False'; S7_HMI_Visible := 'False'} : BOOL;   //EPICS Status variable: MonitHealthy
      "HCB-ACH:ODH-O2iM-3_Maint" { S7_HMI_Accessible := 'False'; S7_HMI_Visible := 'False'} : BOOL;   //EPICS Status variable: Maint
      "HCB-ACH:ODH-O2iM-3_MonitWarning" { S7_HMI_Accessible := 'False'; S7_HMI_Visible := 'False'} : BOOL;   //EPICS Status variable: MonitWarning
      "HCB-ACH:ODH-O2iM-3_SysOK" { S7_HMI_Accessible := 'False'; S7_HMI_Visible := 'False'} : BOOL;   //EPICS Status variable: SysOK
      "HCB-ACH:ODH-O2iM-3_WarmUp" { S7_HMI_Accessible := 'False'; S7_HMI_Visible := 'False'} : BOOL;   //EPICS Status variable: WarmUp
      "HCB-ACH:ODH-O2iM-3_ConnLost" { S7_HMI_Accessible := 'False'; S7_HMI_Visible := 'False'} : BOOL;   //EPICS Status variable: ConnLost
      "HCB-ACH:ODH-O2iM-4_O2Level" { S7_HMI_Accessible := 'False'; S7_HMI_Visible := 'False'} : REAL;   //EPICS Status variable: O2Level
      "HCB-ACH:ODH-O2iM-4_ODHAlarm" { S7_HMI_Accessible := 'False'; S7_HMI_Visible := 'False'} : BOOL;   //EPICS Status variable: ODHAlarm
      "HCB-ACH:ODH-O2iM-4_ODHWarning" { S7_HMI_Accessible := 'False'; S7_HMI_Visible := 'False'} : BOOL;   //EPICS Status variable: ODHWarning
      "HCB-ACH:ODH-O2iM-4_MonitHealthy" { S7_HMI_Accessible := 'False'; S7_HMI_Visible := 'False'} : BOOL;   //EPICS Status variable: MonitHealthy
      "HCB-ACH:ODH-O2iM-4_Maint" { S7_HMI_Accessible := 'False'; S7_HMI_Visible := 'False'} : BOOL;   //EPICS Status variable: Maint
      "HCB-ACH:ODH-O2iM-4_MonitWarning" { S7_HMI_Accessible := 'False'; S7_HMI_Visible := 'False'} : BOOL;   //EPICS Status variable: MonitWarning
      "HCB-ACH:ODH-O2iM-4_SysOK" { S7_HMI_Accessible := 'False'; S7_HMI_Visible := 'False'} : BOOL;   //EPICS Status variable: SysOK
      "HCB-ACH:ODH-O2iM-4_WarmUp" { S7_HMI_Accessible := 'False'; S7_HMI_Visible := 'False'} : BOOL;   //EPICS Status variable: WarmUp
      "HCB-ACH:ODH-O2iM-4_ConnLost" { S7_HMI_Accessible := 'False'; S7_HMI_Visible := 'False'} : BOOL;   //EPICS Status variable: ConnLost
      "HCB-ACH:ODH-O2iM-5_O2Level" { S7_HMI_Accessible := 'False'; S7_HMI_Visible := 'False'} : REAL;   //EPICS Status variable: O2Level
      "HCB-ACH:ODH-O2iM-5_ODHAlarm" { S7_HMI_Accessible := 'False'; S7_HMI_Visible := 'False'} : BOOL;   //EPICS Status variable: ODHAlarm
      "HCB-ACH:ODH-O2iM-5_ODHWarning" { S7_HMI_Accessible := 'False'; S7_HMI_Visible := 'False'} : BOOL;   //EPICS Status variable: ODHWarning
      "HCB-ACH:ODH-O2iM-5_MonitHealthy" { S7_HMI_Accessible := 'False'; S7_HMI_Visible := 'False'} : BOOL;   //EPICS Status variable: MonitHealthy
      "HCB-ACH:ODH-O2iM-5_Maint" { S7_HMI_Accessible := 'False'; S7_HMI_Visible := 'False'} : BOOL;   //EPICS Status variable: Maint
      "HCB-ACH:ODH-O2iM-5_MonitWarning" { S7_HMI_Accessible := 'False'; S7_HMI_Visible := 'False'} : BOOL;   //EPICS Status variable: MonitWarning
      "HCB-ACH:ODH-O2iM-5_SysOK" { S7_HMI_Accessible := 'False'; S7_HMI_Visible := 'False'} : BOOL;   //EPICS Status variable: SysOK
      "HCB-ACH:ODH-O2iM-5_WarmUp" { S7_HMI_Accessible := 'False'; S7_HMI_Visible := 'False'} : BOOL;   //EPICS Status variable: WarmUp
      "HCB-ACH:ODH-O2iM-5_ConnLost" { S7_HMI_Accessible := 'False'; S7_HMI_Visible := 'False'} : BOOL;   //EPICS Status variable: ConnLost
      "HCB-DogSh:ODH-O2iM-12_O2Level" { S7_HMI_Accessible := 'False'; S7_HMI_Visible := 'False'} : REAL;   //EPICS Status variable: O2Level
      "HCB-DogSh:ODH-O2iM-12_ODHAlarm" { S7_HMI_Accessible := 'False'; S7_HMI_Visible := 'False'} : BOOL;   //EPICS Status variable: ODHAlarm
      "HCB-DogSh:ODH-O2iM-12_ODHWarning" { S7_HMI_Accessible := 'False'; S7_HMI_Visible := 'False'} : BOOL;   //EPICS Status variable: ODHWarning
      "HCB-DogSh:ODH-O2iM-12_MonitHealthy" { S7_HMI_Accessible := 'False'; S7_HMI_Visible := 'False'} : BOOL;   //EPICS Status variable: MonitHealthy
      "HCB-DogSh:ODH-O2iM-12_Maint" { S7_HMI_Accessible := 'False'; S7_HMI_Visible := 'False'} : BOOL;   //EPICS Status variable: Maint
      "HCB-DogSh:ODH-O2iM-12_MonitWarning" { S7_HMI_Accessible := 'False'; S7_HMI_Visible := 'False'} : BOOL;   //EPICS Status variable: MonitWarning
      "HCB-DogSh:ODH-O2iM-12_SysOK" { S7_HMI_Accessible := 'False'; S7_HMI_Visible := 'False'} : BOOL;   //EPICS Status variable: SysOK
      "HCB-DogSh:ODH-O2iM-12_WarmUp" { S7_HMI_Accessible := 'False'; S7_HMI_Visible := 'False'} : BOOL;   //EPICS Status variable: WarmUp
      "HCB-DogSh:ODH-O2iM-12_ConnLost" { S7_HMI_Accessible := 'False'; S7_HMI_Visible := 'False'} : BOOL;   //EPICS Status variable: ConnLost
      "HCB-HPGS:ODH-O2iM-10_O2Level" { S7_HMI_Accessible := 'False'; S7_HMI_Visible := 'False'} : REAL;   //EPICS Status variable: O2Level
      "HCB-HPGS:ODH-O2iM-10_ODHAlarm" { S7_HMI_Accessible := 'False'; S7_HMI_Visible := 'False'} : BOOL;   //EPICS Status variable: ODHAlarm
      "HCB-HPGS:ODH-O2iM-10_ODHWarning" { S7_HMI_Accessible := 'False'; S7_HMI_Visible := 'False'} : BOOL;   //EPICS Status variable: ODHWarning
      "HCB-HPGS:ODH-O2iM-10_MonitHealthy" { S7_HMI_Accessible := 'False'; S7_HMI_Visible := 'False'} : BOOL;   //EPICS Status variable: MonitHealthy
      "HCB-HPGS:ODH-O2iM-10_Maint" { S7_HMI_Accessible := 'False'; S7_HMI_Visible := 'False'} : BOOL;   //EPICS Status variable: Maint
      "HCB-HPGS:ODH-O2iM-10_MonitWarning" { S7_HMI_Accessible := 'False'; S7_HMI_Visible := 'False'} : BOOL;   //EPICS Status variable: MonitWarning
      "HCB-HPGS:ODH-O2iM-10_SysOK" { S7_HMI_Accessible := 'False'; S7_HMI_Visible := 'False'} : BOOL;   //EPICS Status variable: SysOK
      "HCB-HPGS:ODH-O2iM-10_WarmUp" { S7_HMI_Accessible := 'False'; S7_HMI_Visible := 'False'} : BOOL;   //EPICS Status variable: WarmUp
      "HCB-HPGS:ODH-O2iM-10_ConnLost" { S7_HMI_Accessible := 'False'; S7_HMI_Visible := 'False'} : BOOL;   //EPICS Status variable: ConnLost
      "HCB-HPGS:ODH-O2iM-11_O2Level" { S7_HMI_Accessible := 'False'; S7_HMI_Visible := 'False'} : REAL;   //EPICS Status variable: O2Level
      "HCB-HPGS:ODH-O2iM-11_ODHAlarm" { S7_HMI_Accessible := 'False'; S7_HMI_Visible := 'False'} : BOOL;   //EPICS Status variable: ODHAlarm
      "HCB-HPGS:ODH-O2iM-11_ODHWarning" { S7_HMI_Accessible := 'False'; S7_HMI_Visible := 'False'} : BOOL;   //EPICS Status variable: ODHWarning
      "HCB-HPGS:ODH-O2iM-11_MonitHealthy" { S7_HMI_Accessible := 'False'; S7_HMI_Visible := 'False'} : BOOL;   //EPICS Status variable: MonitHealthy
      "HCB-HPGS:ODH-O2iM-11_Maint" { S7_HMI_Accessible := 'False'; S7_HMI_Visible := 'False'} : BOOL;   //EPICS Status variable: Maint
      "HCB-HPGS:ODH-O2iM-11_MonitWarning" { S7_HMI_Accessible := 'False'; S7_HMI_Visible := 'False'} : BOOL;   //EPICS Status variable: MonitWarning
      "HCB-HPGS:ODH-O2iM-11_SysOK" { S7_HMI_Accessible := 'False'; S7_HMI_Visible := 'False'} : BOOL;   //EPICS Status variable: SysOK
      "HCB-HPGS:ODH-O2iM-11_WarmUp" { S7_HMI_Accessible := 'False'; S7_HMI_Visible := 'False'} : BOOL;   //EPICS Status variable: WarmUp
      "HCB-HPGS:ODH-O2iM-11_ConnLost" { S7_HMI_Accessible := 'False'; S7_HMI_Visible := 'False'} : BOOL;   //EPICS Status variable: ConnLost
      "HCB-TCH:ODH-O2iM-6_O2Level" { S7_HMI_Accessible := 'False'; S7_HMI_Visible := 'False'} : REAL;   //EPICS Status variable: O2Level
      "HCB-TCH:ODH-O2iM-6_ODHAlarm" { S7_HMI_Accessible := 'False'; S7_HMI_Visible := 'False'} : BOOL;   //EPICS Status variable: ODHAlarm
      "HCB-TCH:ODH-O2iM-6_ODHWarning" { S7_HMI_Accessible := 'False'; S7_HMI_Visible := 'False'} : BOOL;   //EPICS Status variable: ODHWarning
      "HCB-TCH:ODH-O2iM-6_MonitHealthy" { S7_HMI_Accessible := 'False'; S7_HMI_Visible := 'False'} : BOOL;   //EPICS Status variable: MonitHealthy
      "HCB-TCH:ODH-O2iM-6_Maint" { S7_HMI_Accessible := 'False'; S7_HMI_Visible := 'False'} : BOOL;   //EPICS Status variable: Maint
      "HCB-TCH:ODH-O2iM-6_MonitWarning" { S7_HMI_Accessible := 'False'; S7_HMI_Visible := 'False'} : BOOL;   //EPICS Status variable: MonitWarning
      "HCB-TCH:ODH-O2iM-6_SysOK" { S7_HMI_Accessible := 'False'; S7_HMI_Visible := 'False'} : BOOL;   //EPICS Status variable: SysOK
      "HCB-TCH:ODH-O2iM-6_WarmUp" { S7_HMI_Accessible := 'False'; S7_HMI_Visible := 'False'} : BOOL;   //EPICS Status variable: WarmUp
      "HCB-TCH:ODH-O2iM-6_ConnLost" { S7_HMI_Accessible := 'False'; S7_HMI_Visible := 'False'} : BOOL;   //EPICS Status variable: ConnLost
      "HCB-TCH:ODH-O2iM-7_O2Level" { S7_HMI_Accessible := 'False'; S7_HMI_Visible := 'False'} : REAL;   //EPICS Status variable: O2Level
      "HCB-TCH:ODH-O2iM-7_ODHAlarm" { S7_HMI_Accessible := 'False'; S7_HMI_Visible := 'False'} : BOOL;   //EPICS Status variable: ODHAlarm
      "HCB-TCH:ODH-O2iM-7_ODHWarning" { S7_HMI_Accessible := 'False'; S7_HMI_Visible := 'False'} : BOOL;   //EPICS Status variable: ODHWarning
      "HCB-TCH:ODH-O2iM-7_MonitHealthy" { S7_HMI_Accessible := 'False'; S7_HMI_Visible := 'False'} : BOOL;   //EPICS Status variable: MonitHealthy
      "HCB-TCH:ODH-O2iM-7_Maint" { S7_HMI_Accessible := 'False'; S7_HMI_Visible := 'False'} : BOOL;   //EPICS Status variable: Maint
      "HCB-TCH:ODH-O2iM-7_MonitWarning" { S7_HMI_Accessible := 'False'; S7_HMI_Visible := 'False'} : BOOL;   //EPICS Status variable: MonitWarning
      "HCB-TCH:ODH-O2iM-7_SysOK" { S7_HMI_Accessible := 'False'; S7_HMI_Visible := 'False'} : BOOL;   //EPICS Status variable: SysOK
      "HCB-TCH:ODH-O2iM-7_WarmUp" { S7_HMI_Accessible := 'False'; S7_HMI_Visible := 'False'} : BOOL;   //EPICS Status variable: WarmUp
      "HCB-TCH:ODH-O2iM-7_ConnLost" { S7_HMI_Accessible := 'False'; S7_HMI_Visible := 'False'} : BOOL;   //EPICS Status variable: ConnLost
      "HCB-TCH:ODH-O2iM-8_O2Level" { S7_HMI_Accessible := 'False'; S7_HMI_Visible := 'False'} : REAL;   //EPICS Status variable: O2Level
      "HCB-TCH:ODH-O2iM-8_ODHAlarm" { S7_HMI_Accessible := 'False'; S7_HMI_Visible := 'False'} : BOOL;   //EPICS Status variable: ODHAlarm
      "HCB-TCH:ODH-O2iM-8_ODHWarning" { S7_HMI_Accessible := 'False'; S7_HMI_Visible := 'False'} : BOOL;   //EPICS Status variable: ODHWarning
      "HCB-TCH:ODH-O2iM-8_MonitHealthy" { S7_HMI_Accessible := 'False'; S7_HMI_Visible := 'False'} : BOOL;   //EPICS Status variable: MonitHealthy
      "HCB-TCH:ODH-O2iM-8_Maint" { S7_HMI_Accessible := 'False'; S7_HMI_Visible := 'False'} : BOOL;   //EPICS Status variable: Maint
      "HCB-TCH:ODH-O2iM-8_MonitWarning" { S7_HMI_Accessible := 'False'; S7_HMI_Visible := 'False'} : BOOL;   //EPICS Status variable: MonitWarning
      "HCB-TCH:ODH-O2iM-8_SysOK" { S7_HMI_Accessible := 'False'; S7_HMI_Visible := 'False'} : BOOL;   //EPICS Status variable: SysOK
      "HCB-TCH:ODH-O2iM-8_WarmUp" { S7_HMI_Accessible := 'False'; S7_HMI_Visible := 'False'} : BOOL;   //EPICS Status variable: WarmUp
      "HCB-TCH:ODH-O2iM-8_ConnLost" { S7_HMI_Accessible := 'False'; S7_HMI_Visible := 'False'} : BOOL;   //EPICS Status variable: ConnLost
      "HCB-TCH:ODH-O2iM-9_O2Level" { S7_HMI_Accessible := 'False'; S7_HMI_Visible := 'False'} : REAL;   //EPICS Status variable: O2Level
      "HCB-TCH:ODH-O2iM-9_ODHAlarm" { S7_HMI_Accessible := 'False'; S7_HMI_Visible := 'False'} : BOOL;   //EPICS Status variable: ODHAlarm
      "HCB-TCH:ODH-O2iM-9_ODHWarning" { S7_HMI_Accessible := 'False'; S7_HMI_Visible := 'False'} : BOOL;   //EPICS Status variable: ODHWarning
      "HCB-TCH:ODH-O2iM-9_MonitHealthy" { S7_HMI_Accessible := 'False'; S7_HMI_Visible := 'False'} : BOOL;   //EPICS Status variable: MonitHealthy
      "HCB-TCH:ODH-O2iM-9_Maint" { S7_HMI_Accessible := 'False'; S7_HMI_Visible := 'False'} : BOOL;   //EPICS Status variable: Maint
      "HCB-TCH:ODH-O2iM-9_MonitWarning" { S7_HMI_Accessible := 'False'; S7_HMI_Visible := 'False'} : BOOL;   //EPICS Status variable: MonitWarning
      "HCB-TCH:ODH-O2iM-9_SysOK" { S7_HMI_Accessible := 'False'; S7_HMI_Visible := 'False'} : BOOL;   //EPICS Status variable: SysOK
      "HCB-TCH:ODH-O2iM-9_WarmUp" { S7_HMI_Accessible := 'False'; S7_HMI_Visible := 'False'} : BOOL;   //EPICS Status variable: WarmUp
      "HCB-TCH:ODH-O2iM-9_ConnLost" { S7_HMI_Accessible := 'False'; S7_HMI_Visible := 'False'} : BOOL;   //EPICS Status variable: ConnLost
      "CXB-CXH:ODH-RIO-2_SurgeArrOK" { S7_HMI_Accessible := 'False'; S7_HMI_Visible := 'False'} : BOOL;   //EPICS Status variable: SurgeArrOK
      "CXB-CXH:ODH-RIO-2_PS24vOK" { S7_HMI_Accessible := 'False'; S7_HMI_Visible := 'False'} : BOOL;   //EPICS Status variable: PS24vOK
      "CXB-CXH:ODH-RIO-2_UPSBatOK" { S7_HMI_Accessible := 'False'; S7_HMI_Visible := 'False'} : BOOL;   //EPICS Status variable: UPSBatOK
      "CXB-CXH:ODH-RIO-2_UPS24vOK" { S7_HMI_Accessible := 'False'; S7_HMI_Visible := 'False'} : BOOL;   //EPICS Status variable: UPS24vOK
      "CXB-CXH:ODH-RIO-2_UPSBuffReady" { S7_HMI_Accessible := 'False'; S7_HMI_Visible := 'False'} : BOOL;   //EPICS Status variable: UPSBuffReady
      "CXB-CXH:ODH-RIO-2_UPSBatt85" { S7_HMI_Accessible := 'False'; S7_HMI_Visible := 'False'} : BOOL;   //EPICS Status variable: UPSBatt85
      "CXB-CXH:ODH-RIO-2_UPSAlarm" { S7_HMI_Accessible := 'False'; S7_HMI_Visible := 'False'} : BOOL;   //EPICS Status variable: UPSAlarm
      "HCB-ACH:ODH-RIO-1_SurgeArrOK" { S7_HMI_Accessible := 'False'; S7_HMI_Visible := 'False'} : BOOL;   //EPICS Status variable: SurgeArrOK
      "HCB-ACH:ODH-RIO-1_PS24vOK" { S7_HMI_Accessible := 'False'; S7_HMI_Visible := 'False'} : BOOL;   //EPICS Status variable: PS24vOK
      "HCB-ACH:ODH-RIO-1_UPSBatOK" { S7_HMI_Accessible := 'False'; S7_HMI_Visible := 'False'} : BOOL;   //EPICS Status variable: UPSBatOK
      "HCB-ACH:ODH-RIO-1_UPS24vOK" { S7_HMI_Accessible := 'False'; S7_HMI_Visible := 'False'} : BOOL;   //EPICS Status variable: UPS24vOK
      "HCB-ACH:ODH-RIO-1_UPSBuffReady" { S7_HMI_Accessible := 'False'; S7_HMI_Visible := 'False'} : BOOL;   //EPICS Status variable: UPSBuffReady
      "HCB-ACH:ODH-RIO-1_UPSBatt85" { S7_HMI_Accessible := 'False'; S7_HMI_Visible := 'False'} : BOOL;   //EPICS Status variable: UPSBatt85
      "HCB-ACH:ODH-RIO-1_UPSAlarm" { S7_HMI_Accessible := 'False'; S7_HMI_Visible := 'False'} : BOOL;   //EPICS Status variable: UPSAlarm
      "TS2-020Row:CnPw-U-001_SurgeArrOK" { S7_HMI_Accessible := 'False'; S7_HMI_Visible := 'False'} : BOOL;   //EPICS Status variable: SurgeArrOK
      "TS2-020Row:CnPw-U-001_PS24vOK" { S7_HMI_Accessible := 'False'; S7_HMI_Visible := 'False'} : BOOL;   //EPICS Status variable: PS24vOK
      "TS2-020Row:CnPw-U-001_UPSBatOK" { S7_HMI_Accessible := 'False'; S7_HMI_Visible := 'False'} : BOOL;   //EPICS Status variable: UPSBatOK
      "TS2-020Row:CnPw-U-001_UPS24vOK" { S7_HMI_Accessible := 'False'; S7_HMI_Visible := 'False'} : BOOL;   //EPICS Status variable: UPS24vOK
      "TS2-020Row:CnPw-U-001_UPSBuffReady" { S7_HMI_Accessible := 'False'; S7_HMI_Visible := 'False'} : BOOL;   //EPICS Status variable: UPSBuffReady
      "TS2-020Row:CnPw-U-001_UPSBatt85" { S7_HMI_Accessible := 'False'; S7_HMI_Visible := 'False'} : BOOL;   //EPICS Status variable: UPSBatt85
      "TS2-020Row:CnPw-U-001_UPSAlarm" { S7_HMI_Accessible := 'False'; S7_HMI_Visible := 'False'} : BOOL;   //EPICS Status variable: UPSAlarm
   END_STRUCT;
BEGIN
END_DATA_BLOCK
FUNCTION "EPICS_device_calls" : Void
{ S7_Optimized_Access := 'TRUE' }
VERSION : 1.0

   VAR_TEMP
      "CTLG-CS:ODH-Area" : Bool;   // HASH codes are OK
      "CXB-CXH:ODH-Area" : Bool;   // HASH codes are OK
      "CTLG-CS:ODH-O2iM-20" : Bool;   // HASH codes are OK
      "CTLG-CS:ODH-O2iM-21" : Bool;   // HASH codes are OK
      "CTLG-CS:ODH-O2iM-22" : Bool;   // HASH codes are OK
      "CXB-CXH:ODH-O2iM-13" : Bool;   // HASH codes are OK
      "CXB-CXH:ODH-O2iM-14" : Bool;   // HASH codes are OK
      "CXB-CXH:ODH-O2iM-15" : Bool;   // HASH codes are OK
      "CXB-CXH:ODH-O2iM-16" : Bool;   // HASH codes are OK
      "CXB-CXH:ODH-O2iM-17" : Bool;   // HASH codes are OK
      "CXB-CXH:ODH-O2iM-18" : Bool;   // HASH codes are OK
      "CXB-CXH:ODH-O2iM-19" : Bool;   // HASH codes are OK
      "HCB-ACH:ODH-O2iM-1" : Bool;   // HASH codes are OK
      "HCB-ACH:ODH-O2iM-2" : Bool;   // HASH codes are OK
      "HCB-ACH:ODH-O2iM-3" : Bool;   // HASH codes are OK
      "HCB-ACH:ODH-O2iM-4" : Bool;   // HASH codes are OK
      "HCB-ACH:ODH-O2iM-5" : Bool;   // HASH codes are OK
      "HCB-DogSh:ODH-O2iM-12" : Bool;   // HASH codes are OK
      "HCB-HPGS:ODH-O2iM-10" : Bool;   // HASH codes are OK
      "HCB-HPGS:ODH-O2iM-11" : Bool;   // HASH codes are OK
      "HCB-TCH:ODH-O2iM-6" : Bool;   // HASH codes are OK
      "HCB-TCH:ODH-O2iM-7" : Bool;   // HASH codes are OK
      "HCB-TCH:ODH-O2iM-8" : Bool;   // HASH codes are OK
      "HCB-TCH:ODH-O2iM-9" : Bool;   // HASH codes are OK
      "CXB-CXH:ODH-RIO-2" : Bool;   // HASH codes are OK
      "HCB-ACH:ODH-RIO-1" : Bool;   // HASH codes are OK
      "TS2-020Row:CnPw-U-001" : Bool;   // HASH codes are OK
   END_VAR

BEGIN
      //Author: Miklos Boros (miklos.boros@esss.se), Copyrigth 2017-2018 by European Spallation Source, Lund
      //This block was generated by PLCFactory
      //According to HASH:733470530
      //Description: Description: This function calls the devices according to the corresponding device type

        //DO NOT Modify the following line!!!
        "Utilities".TestInProgress := FALSE;


        //********************************************
        // Device name: CTLG-CS:ODH-Area
        // Device type: ODH_Area
        //********************************************

      "DEV_CTLG-CS:ODH-Area_iDB" ();

        //********************************************
        // Device name: CXB-CXH:ODH-Area
        // Device type: ODH_Area
        //********************************************

      "DEV_CXB-CXH:ODH-Area_iDB" ();

        //********************************************
        // Device name: CTLG-CS:ODH-O2iM-20
        // Device type: ODH_O2iM
        //********************************************

      "DEV_CTLG-CS:ODH-O2iM-20_iDB" ();

        //********************************************
        // Device name: CTLG-CS:ODH-O2iM-21
        // Device type: ODH_O2iM
        //********************************************

      "DEV_CTLG-CS:ODH-O2iM-21_iDB" ();

        //********************************************
        // Device name: CTLG-CS:ODH-O2iM-22
        // Device type: ODH_O2iM
        //********************************************

      "DEV_CTLG-CS:ODH-O2iM-22_iDB" ();

        //********************************************
        // Device name: CXB-CXH:ODH-O2iM-13
        // Device type: ODH_O2iM
        //********************************************

      "DEV_CXB-CXH:ODH-O2iM-13_iDB" ();

        //********************************************
        // Device name: CXB-CXH:ODH-O2iM-14
        // Device type: ODH_O2iM
        //********************************************

      "DEV_CXB-CXH:ODH-O2iM-14_iDB" ();

        //********************************************
        // Device name: CXB-CXH:ODH-O2iM-15
        // Device type: ODH_O2iM
        //********************************************

      "DEV_CXB-CXH:ODH-O2iM-15_iDB" ();

        //********************************************
        // Device name: CXB-CXH:ODH-O2iM-16
        // Device type: ODH_O2iM
        //********************************************

      "DEV_CXB-CXH:ODH-O2iM-16_iDB" ();

        //********************************************
        // Device name: CXB-CXH:ODH-O2iM-17
        // Device type: ODH_O2iM
        //********************************************

      "DEV_CXB-CXH:ODH-O2iM-17_iDB" ();

        //********************************************
        // Device name: CXB-CXH:ODH-O2iM-18
        // Device type: ODH_O2iM
        //********************************************

      "DEV_CXB-CXH:ODH-O2iM-18_iDB" ();

        //********************************************
        // Device name: CXB-CXH:ODH-O2iM-19
        // Device type: ODH_O2iM
        //********************************************

      "DEV_CXB-CXH:ODH-O2iM-19_iDB" ();

        //********************************************
        // Device name: HCB-ACH:ODH-O2iM-1
        // Device type: ODH_O2iM
        //********************************************

      "DEV_HCB-ACH:ODH-O2iM-1_iDB" ();

        //********************************************
        // Device name: HCB-ACH:ODH-O2iM-2
        // Device type: ODH_O2iM
        //********************************************

      "DEV_HCB-ACH:ODH-O2iM-2_iDB" ();

        //********************************************
        // Device name: HCB-ACH:ODH-O2iM-3
        // Device type: ODH_O2iM
        //********************************************

      "DEV_HCB-ACH:ODH-O2iM-3_iDB" ();

        //********************************************
        // Device name: HCB-ACH:ODH-O2iM-4
        // Device type: ODH_O2iM
        //********************************************

      "DEV_HCB-ACH:ODH-O2iM-4_iDB" ();

        //********************************************
        // Device name: HCB-ACH:ODH-O2iM-5
        // Device type: ODH_O2iM
        //********************************************

      "DEV_HCB-ACH:ODH-O2iM-5_iDB" ();

        //********************************************
        // Device name: HCB-DogSh:ODH-O2iM-12
        // Device type: ODH_O2iM
        //********************************************

      "DEV_HCB-DogSh:ODH-O2iM-12_iDB" ();

        //********************************************
        // Device name: HCB-HPGS:ODH-O2iM-10
        // Device type: ODH_O2iM
        //********************************************

      "DEV_HCB-HPGS:ODH-O2iM-10_iDB" ();

        //********************************************
        // Device name: HCB-HPGS:ODH-O2iM-11
        // Device type: ODH_O2iM
        //********************************************

      "DEV_HCB-HPGS:ODH-O2iM-11_iDB" ();

        //********************************************
        // Device name: HCB-TCH:ODH-O2iM-6
        // Device type: ODH_O2iM
        //********************************************

      "DEV_HCB-TCH:ODH-O2iM-6_iDB" ();

        //********************************************
        // Device name: HCB-TCH:ODH-O2iM-7
        // Device type: ODH_O2iM
        //********************************************

      "DEV_HCB-TCH:ODH-O2iM-7_iDB" ();

        //********************************************
        // Device name: HCB-TCH:ODH-O2iM-8
        // Device type: ODH_O2iM
        //********************************************

      "DEV_HCB-TCH:ODH-O2iM-8_iDB" ();

        //********************************************
        // Device name: HCB-TCH:ODH-O2iM-9
        // Device type: ODH_O2iM
        //********************************************

      "DEV_HCB-TCH:ODH-O2iM-9_iDB" ();

        //********************************************
        // Device name: CXB-CXH:ODH-RIO-2
        // Device type: ODH_Rack
        //********************************************

      "DEV_CXB-CXH:ODH-RIO-2_iDB" ();

        //********************************************
        // Device name: HCB-ACH:ODH-RIO-1
        // Device type: ODH_Rack
        //********************************************

      "DEV_HCB-ACH:ODH-RIO-1_iDB" ();

        //********************************************
        // Device name: TS2-020Row:CnPw-U-001
        // Device type: ODH_Rack
        //********************************************

      "DEV_TS2-020Row:CnPw-U-001_iDB" ();
END_FUNCTION
FUNCTION "EPICS_device_calls_test" : Void
{ S7_Optimized_Access := 'TRUE' }
VERSION : 1.0

   VAR_TEMP
      "CTLG-CS:ODH-Area" : Bool;   // HASH codes are OK
      "CXB-CXH:ODH-Area" : Bool;   // HASH codes are OK
      "CTLG-CS:ODH-O2iM-20" : Bool;   // HASH codes are OK
      "CTLG-CS:ODH-O2iM-21" : Bool;   // HASH codes are OK
      "CTLG-CS:ODH-O2iM-22" : Bool;   // HASH codes are OK
      "CXB-CXH:ODH-O2iM-13" : Bool;   // HASH codes are OK
      "CXB-CXH:ODH-O2iM-14" : Bool;   // HASH codes are OK
      "CXB-CXH:ODH-O2iM-15" : Bool;   // HASH codes are OK
      "CXB-CXH:ODH-O2iM-16" : Bool;   // HASH codes are OK
      "CXB-CXH:ODH-O2iM-17" : Bool;   // HASH codes are OK
      "CXB-CXH:ODH-O2iM-18" : Bool;   // HASH codes are OK
      "CXB-CXH:ODH-O2iM-19" : Bool;   // HASH codes are OK
      "HCB-ACH:ODH-O2iM-1" : Bool;   // HASH codes are OK
      "HCB-ACH:ODH-O2iM-2" : Bool;   // HASH codes are OK
      "HCB-ACH:ODH-O2iM-3" : Bool;   // HASH codes are OK
      "HCB-ACH:ODH-O2iM-4" : Bool;   // HASH codes are OK
      "HCB-ACH:ODH-O2iM-5" : Bool;   // HASH codes are OK
      "HCB-DogSh:ODH-O2iM-12" : Bool;   // HASH codes are OK
      "HCB-HPGS:ODH-O2iM-10" : Bool;   // HASH codes are OK
      "HCB-HPGS:ODH-O2iM-11" : Bool;   // HASH codes are OK
      "HCB-TCH:ODH-O2iM-6" : Bool;   // HASH codes are OK
      "HCB-TCH:ODH-O2iM-7" : Bool;   // HASH codes are OK
      "HCB-TCH:ODH-O2iM-8" : Bool;   // HASH codes are OK
      "HCB-TCH:ODH-O2iM-9" : Bool;   // HASH codes are OK
      "CXB-CXH:ODH-RIO-2" : Bool;   // HASH codes are OK
      "HCB-ACH:ODH-RIO-1" : Bool;   // HASH codes are OK
      "TS2-020Row:CnPw-U-001" : Bool;   // HASH codes are OK
   END_VAR

BEGIN
      //Author: Miklos Boros (miklos.boros@esss.se), Copyrigth 2017-2018 by European Spallation Source, Lund
      //This block was generated by PLCFactory
      //According to HASH:733470530
      //Description: Description: This function calls the devices according to the corresponding device type

      //DO NOT Modify the following line!!!
      "Utilities".TestInProgress := TRUE;


      //********************************************
      // Device name: CTLG-CS:ODH-Area
      // Device type: ODH_Area
      //********************************************

      "DEV_CTLG-CS:ODH-Area_iDB" (
                                 "Alarm" := "EPICS_PLC_Tester".#"CTLG-CS:ODH-Area_Alarm",
                                 "WarmUp" := "EPICS_PLC_Tester".#"CTLG-CS:ODH-Area_WarmUp",
                                 "ConnLost" := "EPICS_PLC_Tester".#"CTLG-CS:ODH-Area_ConnLost",
                                 DEVICE_PARAM_OK=>#"CTLG-CS:ODH-Area");

      //********************************************
      // Device name: CXB-CXH:ODH-Area
      // Device type: ODH_Area
      //********************************************

      "DEV_CXB-CXH:ODH-Area_iDB" (
                                 "Alarm" := "EPICS_PLC_Tester".#"CXB-CXH:ODH-Area_Alarm",
                                 "WarmUp" := "EPICS_PLC_Tester".#"CXB-CXH:ODH-Area_WarmUp",
                                 "ConnLost" := "EPICS_PLC_Tester".#"CXB-CXH:ODH-Area_ConnLost",
                                 DEVICE_PARAM_OK=>#"CXB-CXH:ODH-Area");

      //********************************************
      // Device name: CTLG-CS:ODH-O2iM-20
      // Device type: ODH_O2iM
      //********************************************

      "DEV_CTLG-CS:ODH-O2iM-20_iDB" (
                                 "O2Level" := "EPICS_PLC_Tester".#"CTLG-CS:ODH-O2iM-20_O2Level",
                                 "ODHAlarm" := "EPICS_PLC_Tester".#"CTLG-CS:ODH-O2iM-20_ODHAlarm",
                                 "ODHWarning" := "EPICS_PLC_Tester".#"CTLG-CS:ODH-O2iM-20_ODHWarning",
                                 "MonitHealthy" := "EPICS_PLC_Tester".#"CTLG-CS:ODH-O2iM-20_MonitHealthy",
                                 "Maint" := "EPICS_PLC_Tester".#"CTLG-CS:ODH-O2iM-20_Maint",
                                 "MonitWarning" := "EPICS_PLC_Tester".#"CTLG-CS:ODH-O2iM-20_MonitWarning",
                                 "SysOK" := "EPICS_PLC_Tester".#"CTLG-CS:ODH-O2iM-20_SysOK",
                                 "WarmUp" := "EPICS_PLC_Tester".#"CTLG-CS:ODH-O2iM-20_WarmUp",
                                 "ConnLost" := "EPICS_PLC_Tester".#"CTLG-CS:ODH-O2iM-20_ConnLost",
                                 DEVICE_PARAM_OK=>#"CTLG-CS:ODH-O2iM-20");

      //********************************************
      // Device name: CTLG-CS:ODH-O2iM-21
      // Device type: ODH_O2iM
      //********************************************

      "DEV_CTLG-CS:ODH-O2iM-21_iDB" (
                                 "O2Level" := "EPICS_PLC_Tester".#"CTLG-CS:ODH-O2iM-21_O2Level",
                                 "ODHAlarm" := "EPICS_PLC_Tester".#"CTLG-CS:ODH-O2iM-21_ODHAlarm",
                                 "ODHWarning" := "EPICS_PLC_Tester".#"CTLG-CS:ODH-O2iM-21_ODHWarning",
                                 "MonitHealthy" := "EPICS_PLC_Tester".#"CTLG-CS:ODH-O2iM-21_MonitHealthy",
                                 "Maint" := "EPICS_PLC_Tester".#"CTLG-CS:ODH-O2iM-21_Maint",
                                 "MonitWarning" := "EPICS_PLC_Tester".#"CTLG-CS:ODH-O2iM-21_MonitWarning",
                                 "SysOK" := "EPICS_PLC_Tester".#"CTLG-CS:ODH-O2iM-21_SysOK",
                                 "WarmUp" := "EPICS_PLC_Tester".#"CTLG-CS:ODH-O2iM-21_WarmUp",
                                 "ConnLost" := "EPICS_PLC_Tester".#"CTLG-CS:ODH-O2iM-21_ConnLost",
                                 DEVICE_PARAM_OK=>#"CTLG-CS:ODH-O2iM-21");

      //********************************************
      // Device name: CTLG-CS:ODH-O2iM-22
      // Device type: ODH_O2iM
      //********************************************

      "DEV_CTLG-CS:ODH-O2iM-22_iDB" (
                                 "O2Level" := "EPICS_PLC_Tester".#"CTLG-CS:ODH-O2iM-22_O2Level",
                                 "ODHAlarm" := "EPICS_PLC_Tester".#"CTLG-CS:ODH-O2iM-22_ODHAlarm",
                                 "ODHWarning" := "EPICS_PLC_Tester".#"CTLG-CS:ODH-O2iM-22_ODHWarning",
                                 "MonitHealthy" := "EPICS_PLC_Tester".#"CTLG-CS:ODH-O2iM-22_MonitHealthy",
                                 "Maint" := "EPICS_PLC_Tester".#"CTLG-CS:ODH-O2iM-22_Maint",
                                 "MonitWarning" := "EPICS_PLC_Tester".#"CTLG-CS:ODH-O2iM-22_MonitWarning",
                                 "SysOK" := "EPICS_PLC_Tester".#"CTLG-CS:ODH-O2iM-22_SysOK",
                                 "WarmUp" := "EPICS_PLC_Tester".#"CTLG-CS:ODH-O2iM-22_WarmUp",
                                 "ConnLost" := "EPICS_PLC_Tester".#"CTLG-CS:ODH-O2iM-22_ConnLost",
                                 DEVICE_PARAM_OK=>#"CTLG-CS:ODH-O2iM-22");

      //********************************************
      // Device name: CXB-CXH:ODH-O2iM-13
      // Device type: ODH_O2iM
      //********************************************

      "DEV_CXB-CXH:ODH-O2iM-13_iDB" (
                                 "O2Level" := "EPICS_PLC_Tester".#"CXB-CXH:ODH-O2iM-13_O2Level",
                                 "ODHAlarm" := "EPICS_PLC_Tester".#"CXB-CXH:ODH-O2iM-13_ODHAlarm",
                                 "ODHWarning" := "EPICS_PLC_Tester".#"CXB-CXH:ODH-O2iM-13_ODHWarning",
                                 "MonitHealthy" := "EPICS_PLC_Tester".#"CXB-CXH:ODH-O2iM-13_MonitHealthy",
                                 "Maint" := "EPICS_PLC_Tester".#"CXB-CXH:ODH-O2iM-13_Maint",
                                 "MonitWarning" := "EPICS_PLC_Tester".#"CXB-CXH:ODH-O2iM-13_MonitWarning",
                                 "SysOK" := "EPICS_PLC_Tester".#"CXB-CXH:ODH-O2iM-13_SysOK",
                                 "WarmUp" := "EPICS_PLC_Tester".#"CXB-CXH:ODH-O2iM-13_WarmUp",
                                 "ConnLost" := "EPICS_PLC_Tester".#"CXB-CXH:ODH-O2iM-13_ConnLost",
                                 DEVICE_PARAM_OK=>#"CXB-CXH:ODH-O2iM-13");

      //********************************************
      // Device name: CXB-CXH:ODH-O2iM-14
      // Device type: ODH_O2iM
      //********************************************

      "DEV_CXB-CXH:ODH-O2iM-14_iDB" (
                                 "O2Level" := "EPICS_PLC_Tester".#"CXB-CXH:ODH-O2iM-14_O2Level",
                                 "ODHAlarm" := "EPICS_PLC_Tester".#"CXB-CXH:ODH-O2iM-14_ODHAlarm",
                                 "ODHWarning" := "EPICS_PLC_Tester".#"CXB-CXH:ODH-O2iM-14_ODHWarning",
                                 "MonitHealthy" := "EPICS_PLC_Tester".#"CXB-CXH:ODH-O2iM-14_MonitHealthy",
                                 "Maint" := "EPICS_PLC_Tester".#"CXB-CXH:ODH-O2iM-14_Maint",
                                 "MonitWarning" := "EPICS_PLC_Tester".#"CXB-CXH:ODH-O2iM-14_MonitWarning",
                                 "SysOK" := "EPICS_PLC_Tester".#"CXB-CXH:ODH-O2iM-14_SysOK",
                                 "WarmUp" := "EPICS_PLC_Tester".#"CXB-CXH:ODH-O2iM-14_WarmUp",
                                 "ConnLost" := "EPICS_PLC_Tester".#"CXB-CXH:ODH-O2iM-14_ConnLost",
                                 DEVICE_PARAM_OK=>#"CXB-CXH:ODH-O2iM-14");

      //********************************************
      // Device name: CXB-CXH:ODH-O2iM-15
      // Device type: ODH_O2iM
      //********************************************

      "DEV_CXB-CXH:ODH-O2iM-15_iDB" (
                                 "O2Level" := "EPICS_PLC_Tester".#"CXB-CXH:ODH-O2iM-15_O2Level",
                                 "ODHAlarm" := "EPICS_PLC_Tester".#"CXB-CXH:ODH-O2iM-15_ODHAlarm",
                                 "ODHWarning" := "EPICS_PLC_Tester".#"CXB-CXH:ODH-O2iM-15_ODHWarning",
                                 "MonitHealthy" := "EPICS_PLC_Tester".#"CXB-CXH:ODH-O2iM-15_MonitHealthy",
                                 "Maint" := "EPICS_PLC_Tester".#"CXB-CXH:ODH-O2iM-15_Maint",
                                 "MonitWarning" := "EPICS_PLC_Tester".#"CXB-CXH:ODH-O2iM-15_MonitWarning",
                                 "SysOK" := "EPICS_PLC_Tester".#"CXB-CXH:ODH-O2iM-15_SysOK",
                                 "WarmUp" := "EPICS_PLC_Tester".#"CXB-CXH:ODH-O2iM-15_WarmUp",
                                 "ConnLost" := "EPICS_PLC_Tester".#"CXB-CXH:ODH-O2iM-15_ConnLost",
                                 DEVICE_PARAM_OK=>#"CXB-CXH:ODH-O2iM-15");

      //********************************************
      // Device name: CXB-CXH:ODH-O2iM-16
      // Device type: ODH_O2iM
      //********************************************

      "DEV_CXB-CXH:ODH-O2iM-16_iDB" (
                                 "O2Level" := "EPICS_PLC_Tester".#"CXB-CXH:ODH-O2iM-16_O2Level",
                                 "ODHAlarm" := "EPICS_PLC_Tester".#"CXB-CXH:ODH-O2iM-16_ODHAlarm",
                                 "ODHWarning" := "EPICS_PLC_Tester".#"CXB-CXH:ODH-O2iM-16_ODHWarning",
                                 "MonitHealthy" := "EPICS_PLC_Tester".#"CXB-CXH:ODH-O2iM-16_MonitHealthy",
                                 "Maint" := "EPICS_PLC_Tester".#"CXB-CXH:ODH-O2iM-16_Maint",
                                 "MonitWarning" := "EPICS_PLC_Tester".#"CXB-CXH:ODH-O2iM-16_MonitWarning",
                                 "SysOK" := "EPICS_PLC_Tester".#"CXB-CXH:ODH-O2iM-16_SysOK",
                                 "WarmUp" := "EPICS_PLC_Tester".#"CXB-CXH:ODH-O2iM-16_WarmUp",
                                 "ConnLost" := "EPICS_PLC_Tester".#"CXB-CXH:ODH-O2iM-16_ConnLost",
                                 DEVICE_PARAM_OK=>#"CXB-CXH:ODH-O2iM-16");

      //********************************************
      // Device name: CXB-CXH:ODH-O2iM-17
      // Device type: ODH_O2iM
      //********************************************

      "DEV_CXB-CXH:ODH-O2iM-17_iDB" (
                                 "O2Level" := "EPICS_PLC_Tester".#"CXB-CXH:ODH-O2iM-17_O2Level",
                                 "ODHAlarm" := "EPICS_PLC_Tester".#"CXB-CXH:ODH-O2iM-17_ODHAlarm",
                                 "ODHWarning" := "EPICS_PLC_Tester".#"CXB-CXH:ODH-O2iM-17_ODHWarning",
                                 "MonitHealthy" := "EPICS_PLC_Tester".#"CXB-CXH:ODH-O2iM-17_MonitHealthy",
                                 "Maint" := "EPICS_PLC_Tester".#"CXB-CXH:ODH-O2iM-17_Maint",
                                 "MonitWarning" := "EPICS_PLC_Tester".#"CXB-CXH:ODH-O2iM-17_MonitWarning",
                                 "SysOK" := "EPICS_PLC_Tester".#"CXB-CXH:ODH-O2iM-17_SysOK",
                                 "WarmUp" := "EPICS_PLC_Tester".#"CXB-CXH:ODH-O2iM-17_WarmUp",
                                 "ConnLost" := "EPICS_PLC_Tester".#"CXB-CXH:ODH-O2iM-17_ConnLost",
                                 DEVICE_PARAM_OK=>#"CXB-CXH:ODH-O2iM-17");

      //********************************************
      // Device name: CXB-CXH:ODH-O2iM-18
      // Device type: ODH_O2iM
      //********************************************

      "DEV_CXB-CXH:ODH-O2iM-18_iDB" (
                                 "O2Level" := "EPICS_PLC_Tester".#"CXB-CXH:ODH-O2iM-18_O2Level",
                                 "ODHAlarm" := "EPICS_PLC_Tester".#"CXB-CXH:ODH-O2iM-18_ODHAlarm",
                                 "ODHWarning" := "EPICS_PLC_Tester".#"CXB-CXH:ODH-O2iM-18_ODHWarning",
                                 "MonitHealthy" := "EPICS_PLC_Tester".#"CXB-CXH:ODH-O2iM-18_MonitHealthy",
                                 "Maint" := "EPICS_PLC_Tester".#"CXB-CXH:ODH-O2iM-18_Maint",
                                 "MonitWarning" := "EPICS_PLC_Tester".#"CXB-CXH:ODH-O2iM-18_MonitWarning",
                                 "SysOK" := "EPICS_PLC_Tester".#"CXB-CXH:ODH-O2iM-18_SysOK",
                                 "WarmUp" := "EPICS_PLC_Tester".#"CXB-CXH:ODH-O2iM-18_WarmUp",
                                 "ConnLost" := "EPICS_PLC_Tester".#"CXB-CXH:ODH-O2iM-18_ConnLost",
                                 DEVICE_PARAM_OK=>#"CXB-CXH:ODH-O2iM-18");

      //********************************************
      // Device name: CXB-CXH:ODH-O2iM-19
      // Device type: ODH_O2iM
      //********************************************

      "DEV_CXB-CXH:ODH-O2iM-19_iDB" (
                                 "O2Level" := "EPICS_PLC_Tester".#"CXB-CXH:ODH-O2iM-19_O2Level",
                                 "ODHAlarm" := "EPICS_PLC_Tester".#"CXB-CXH:ODH-O2iM-19_ODHAlarm",
                                 "ODHWarning" := "EPICS_PLC_Tester".#"CXB-CXH:ODH-O2iM-19_ODHWarning",
                                 "MonitHealthy" := "EPICS_PLC_Tester".#"CXB-CXH:ODH-O2iM-19_MonitHealthy",
                                 "Maint" := "EPICS_PLC_Tester".#"CXB-CXH:ODH-O2iM-19_Maint",
                                 "MonitWarning" := "EPICS_PLC_Tester".#"CXB-CXH:ODH-O2iM-19_MonitWarning",
                                 "SysOK" := "EPICS_PLC_Tester".#"CXB-CXH:ODH-O2iM-19_SysOK",
                                 "WarmUp" := "EPICS_PLC_Tester".#"CXB-CXH:ODH-O2iM-19_WarmUp",
                                 "ConnLost" := "EPICS_PLC_Tester".#"CXB-CXH:ODH-O2iM-19_ConnLost",
                                 DEVICE_PARAM_OK=>#"CXB-CXH:ODH-O2iM-19");

      //********************************************
      // Device name: HCB-ACH:ODH-O2iM-1
      // Device type: ODH_O2iM
      //********************************************

      "DEV_HCB-ACH:ODH-O2iM-1_iDB" (
                                 "O2Level" := "EPICS_PLC_Tester".#"HCB-ACH:ODH-O2iM-1_O2Level",
                                 "ODHAlarm" := "EPICS_PLC_Tester".#"HCB-ACH:ODH-O2iM-1_ODHAlarm",
                                 "ODHWarning" := "EPICS_PLC_Tester".#"HCB-ACH:ODH-O2iM-1_ODHWarning",
                                 "MonitHealthy" := "EPICS_PLC_Tester".#"HCB-ACH:ODH-O2iM-1_MonitHealthy",
                                 "Maint" := "EPICS_PLC_Tester".#"HCB-ACH:ODH-O2iM-1_Maint",
                                 "MonitWarning" := "EPICS_PLC_Tester".#"HCB-ACH:ODH-O2iM-1_MonitWarning",
                                 "SysOK" := "EPICS_PLC_Tester".#"HCB-ACH:ODH-O2iM-1_SysOK",
                                 "WarmUp" := "EPICS_PLC_Tester".#"HCB-ACH:ODH-O2iM-1_WarmUp",
                                 "ConnLost" := "EPICS_PLC_Tester".#"HCB-ACH:ODH-O2iM-1_ConnLost",
                                 DEVICE_PARAM_OK=>#"HCB-ACH:ODH-O2iM-1");

      //********************************************
      // Device name: HCB-ACH:ODH-O2iM-2
      // Device type: ODH_O2iM
      //********************************************

      "DEV_HCB-ACH:ODH-O2iM-2_iDB" (
                                 "O2Level" := "EPICS_PLC_Tester".#"HCB-ACH:ODH-O2iM-2_O2Level",
                                 "ODHAlarm" := "EPICS_PLC_Tester".#"HCB-ACH:ODH-O2iM-2_ODHAlarm",
                                 "ODHWarning" := "EPICS_PLC_Tester".#"HCB-ACH:ODH-O2iM-2_ODHWarning",
                                 "MonitHealthy" := "EPICS_PLC_Tester".#"HCB-ACH:ODH-O2iM-2_MonitHealthy",
                                 "Maint" := "EPICS_PLC_Tester".#"HCB-ACH:ODH-O2iM-2_Maint",
                                 "MonitWarning" := "EPICS_PLC_Tester".#"HCB-ACH:ODH-O2iM-2_MonitWarning",
                                 "SysOK" := "EPICS_PLC_Tester".#"HCB-ACH:ODH-O2iM-2_SysOK",
                                 "WarmUp" := "EPICS_PLC_Tester".#"HCB-ACH:ODH-O2iM-2_WarmUp",
                                 "ConnLost" := "EPICS_PLC_Tester".#"HCB-ACH:ODH-O2iM-2_ConnLost",
                                 DEVICE_PARAM_OK=>#"HCB-ACH:ODH-O2iM-2");

      //********************************************
      // Device name: HCB-ACH:ODH-O2iM-3
      // Device type: ODH_O2iM
      //********************************************

      "DEV_HCB-ACH:ODH-O2iM-3_iDB" (
                                 "O2Level" := "EPICS_PLC_Tester".#"HCB-ACH:ODH-O2iM-3_O2Level",
                                 "ODHAlarm" := "EPICS_PLC_Tester".#"HCB-ACH:ODH-O2iM-3_ODHAlarm",
                                 "ODHWarning" := "EPICS_PLC_Tester".#"HCB-ACH:ODH-O2iM-3_ODHWarning",
                                 "MonitHealthy" := "EPICS_PLC_Tester".#"HCB-ACH:ODH-O2iM-3_MonitHealthy",
                                 "Maint" := "EPICS_PLC_Tester".#"HCB-ACH:ODH-O2iM-3_Maint",
                                 "MonitWarning" := "EPICS_PLC_Tester".#"HCB-ACH:ODH-O2iM-3_MonitWarning",
                                 "SysOK" := "EPICS_PLC_Tester".#"HCB-ACH:ODH-O2iM-3_SysOK",
                                 "WarmUp" := "EPICS_PLC_Tester".#"HCB-ACH:ODH-O2iM-3_WarmUp",
                                 "ConnLost" := "EPICS_PLC_Tester".#"HCB-ACH:ODH-O2iM-3_ConnLost",
                                 DEVICE_PARAM_OK=>#"HCB-ACH:ODH-O2iM-3");

      //********************************************
      // Device name: HCB-ACH:ODH-O2iM-4
      // Device type: ODH_O2iM
      //********************************************

      "DEV_HCB-ACH:ODH-O2iM-4_iDB" (
                                 "O2Level" := "EPICS_PLC_Tester".#"HCB-ACH:ODH-O2iM-4_O2Level",
                                 "ODHAlarm" := "EPICS_PLC_Tester".#"HCB-ACH:ODH-O2iM-4_ODHAlarm",
                                 "ODHWarning" := "EPICS_PLC_Tester".#"HCB-ACH:ODH-O2iM-4_ODHWarning",
                                 "MonitHealthy" := "EPICS_PLC_Tester".#"HCB-ACH:ODH-O2iM-4_MonitHealthy",
                                 "Maint" := "EPICS_PLC_Tester".#"HCB-ACH:ODH-O2iM-4_Maint",
                                 "MonitWarning" := "EPICS_PLC_Tester".#"HCB-ACH:ODH-O2iM-4_MonitWarning",
                                 "SysOK" := "EPICS_PLC_Tester".#"HCB-ACH:ODH-O2iM-4_SysOK",
                                 "WarmUp" := "EPICS_PLC_Tester".#"HCB-ACH:ODH-O2iM-4_WarmUp",
                                 "ConnLost" := "EPICS_PLC_Tester".#"HCB-ACH:ODH-O2iM-4_ConnLost",
                                 DEVICE_PARAM_OK=>#"HCB-ACH:ODH-O2iM-4");

      //********************************************
      // Device name: HCB-ACH:ODH-O2iM-5
      // Device type: ODH_O2iM
      //********************************************

      "DEV_HCB-ACH:ODH-O2iM-5_iDB" (
                                 "O2Level" := "EPICS_PLC_Tester".#"HCB-ACH:ODH-O2iM-5_O2Level",
                                 "ODHAlarm" := "EPICS_PLC_Tester".#"HCB-ACH:ODH-O2iM-5_ODHAlarm",
                                 "ODHWarning" := "EPICS_PLC_Tester".#"HCB-ACH:ODH-O2iM-5_ODHWarning",
                                 "MonitHealthy" := "EPICS_PLC_Tester".#"HCB-ACH:ODH-O2iM-5_MonitHealthy",
                                 "Maint" := "EPICS_PLC_Tester".#"HCB-ACH:ODH-O2iM-5_Maint",
                                 "MonitWarning" := "EPICS_PLC_Tester".#"HCB-ACH:ODH-O2iM-5_MonitWarning",
                                 "SysOK" := "EPICS_PLC_Tester".#"HCB-ACH:ODH-O2iM-5_SysOK",
                                 "WarmUp" := "EPICS_PLC_Tester".#"HCB-ACH:ODH-O2iM-5_WarmUp",
                                 "ConnLost" := "EPICS_PLC_Tester".#"HCB-ACH:ODH-O2iM-5_ConnLost",
                                 DEVICE_PARAM_OK=>#"HCB-ACH:ODH-O2iM-5");

      //********************************************
      // Device name: HCB-DogSh:ODH-O2iM-12
      // Device type: ODH_O2iM
      //********************************************

      "DEV_HCB-DogSh:ODH-O2iM-12_iDB" (
                                 "O2Level" := "EPICS_PLC_Tester".#"HCB-DogSh:ODH-O2iM-12_O2Level",
                                 "ODHAlarm" := "EPICS_PLC_Tester".#"HCB-DogSh:ODH-O2iM-12_ODHAlarm",
                                 "ODHWarning" := "EPICS_PLC_Tester".#"HCB-DogSh:ODH-O2iM-12_ODHWarning",
                                 "MonitHealthy" := "EPICS_PLC_Tester".#"HCB-DogSh:ODH-O2iM-12_MonitHealthy",
                                 "Maint" := "EPICS_PLC_Tester".#"HCB-DogSh:ODH-O2iM-12_Maint",
                                 "MonitWarning" := "EPICS_PLC_Tester".#"HCB-DogSh:ODH-O2iM-12_MonitWarning",
                                 "SysOK" := "EPICS_PLC_Tester".#"HCB-DogSh:ODH-O2iM-12_SysOK",
                                 "WarmUp" := "EPICS_PLC_Tester".#"HCB-DogSh:ODH-O2iM-12_WarmUp",
                                 "ConnLost" := "EPICS_PLC_Tester".#"HCB-DogSh:ODH-O2iM-12_ConnLost",
                                 DEVICE_PARAM_OK=>#"HCB-DogSh:ODH-O2iM-12");

      //********************************************
      // Device name: HCB-HPGS:ODH-O2iM-10
      // Device type: ODH_O2iM
      //********************************************

      "DEV_HCB-HPGS:ODH-O2iM-10_iDB" (
                                 "O2Level" := "EPICS_PLC_Tester".#"HCB-HPGS:ODH-O2iM-10_O2Level",
                                 "ODHAlarm" := "EPICS_PLC_Tester".#"HCB-HPGS:ODH-O2iM-10_ODHAlarm",
                                 "ODHWarning" := "EPICS_PLC_Tester".#"HCB-HPGS:ODH-O2iM-10_ODHWarning",
                                 "MonitHealthy" := "EPICS_PLC_Tester".#"HCB-HPGS:ODH-O2iM-10_MonitHealthy",
                                 "Maint" := "EPICS_PLC_Tester".#"HCB-HPGS:ODH-O2iM-10_Maint",
                                 "MonitWarning" := "EPICS_PLC_Tester".#"HCB-HPGS:ODH-O2iM-10_MonitWarning",
                                 "SysOK" := "EPICS_PLC_Tester".#"HCB-HPGS:ODH-O2iM-10_SysOK",
                                 "WarmUp" := "EPICS_PLC_Tester".#"HCB-HPGS:ODH-O2iM-10_WarmUp",
                                 "ConnLost" := "EPICS_PLC_Tester".#"HCB-HPGS:ODH-O2iM-10_ConnLost",
                                 DEVICE_PARAM_OK=>#"HCB-HPGS:ODH-O2iM-10");

      //********************************************
      // Device name: HCB-HPGS:ODH-O2iM-11
      // Device type: ODH_O2iM
      //********************************************

      "DEV_HCB-HPGS:ODH-O2iM-11_iDB" (
                                 "O2Level" := "EPICS_PLC_Tester".#"HCB-HPGS:ODH-O2iM-11_O2Level",
                                 "ODHAlarm" := "EPICS_PLC_Tester".#"HCB-HPGS:ODH-O2iM-11_ODHAlarm",
                                 "ODHWarning" := "EPICS_PLC_Tester".#"HCB-HPGS:ODH-O2iM-11_ODHWarning",
                                 "MonitHealthy" := "EPICS_PLC_Tester".#"HCB-HPGS:ODH-O2iM-11_MonitHealthy",
                                 "Maint" := "EPICS_PLC_Tester".#"HCB-HPGS:ODH-O2iM-11_Maint",
                                 "MonitWarning" := "EPICS_PLC_Tester".#"HCB-HPGS:ODH-O2iM-11_MonitWarning",
                                 "SysOK" := "EPICS_PLC_Tester".#"HCB-HPGS:ODH-O2iM-11_SysOK",
                                 "WarmUp" := "EPICS_PLC_Tester".#"HCB-HPGS:ODH-O2iM-11_WarmUp",
                                 "ConnLost" := "EPICS_PLC_Tester".#"HCB-HPGS:ODH-O2iM-11_ConnLost",
                                 DEVICE_PARAM_OK=>#"HCB-HPGS:ODH-O2iM-11");

      //********************************************
      // Device name: HCB-TCH:ODH-O2iM-6
      // Device type: ODH_O2iM
      //********************************************

      "DEV_HCB-TCH:ODH-O2iM-6_iDB" (
                                 "O2Level" := "EPICS_PLC_Tester".#"HCB-TCH:ODH-O2iM-6_O2Level",
                                 "ODHAlarm" := "EPICS_PLC_Tester".#"HCB-TCH:ODH-O2iM-6_ODHAlarm",
                                 "ODHWarning" := "EPICS_PLC_Tester".#"HCB-TCH:ODH-O2iM-6_ODHWarning",
                                 "MonitHealthy" := "EPICS_PLC_Tester".#"HCB-TCH:ODH-O2iM-6_MonitHealthy",
                                 "Maint" := "EPICS_PLC_Tester".#"HCB-TCH:ODH-O2iM-6_Maint",
                                 "MonitWarning" := "EPICS_PLC_Tester".#"HCB-TCH:ODH-O2iM-6_MonitWarning",
                                 "SysOK" := "EPICS_PLC_Tester".#"HCB-TCH:ODH-O2iM-6_SysOK",
                                 "WarmUp" := "EPICS_PLC_Tester".#"HCB-TCH:ODH-O2iM-6_WarmUp",
                                 "ConnLost" := "EPICS_PLC_Tester".#"HCB-TCH:ODH-O2iM-6_ConnLost",
                                 DEVICE_PARAM_OK=>#"HCB-TCH:ODH-O2iM-6");

      //********************************************
      // Device name: HCB-TCH:ODH-O2iM-7
      // Device type: ODH_O2iM
      //********************************************

      "DEV_HCB-TCH:ODH-O2iM-7_iDB" (
                                 "O2Level" := "EPICS_PLC_Tester".#"HCB-TCH:ODH-O2iM-7_O2Level",
                                 "ODHAlarm" := "EPICS_PLC_Tester".#"HCB-TCH:ODH-O2iM-7_ODHAlarm",
                                 "ODHWarning" := "EPICS_PLC_Tester".#"HCB-TCH:ODH-O2iM-7_ODHWarning",
                                 "MonitHealthy" := "EPICS_PLC_Tester".#"HCB-TCH:ODH-O2iM-7_MonitHealthy",
                                 "Maint" := "EPICS_PLC_Tester".#"HCB-TCH:ODH-O2iM-7_Maint",
                                 "MonitWarning" := "EPICS_PLC_Tester".#"HCB-TCH:ODH-O2iM-7_MonitWarning",
                                 "SysOK" := "EPICS_PLC_Tester".#"HCB-TCH:ODH-O2iM-7_SysOK",
                                 "WarmUp" := "EPICS_PLC_Tester".#"HCB-TCH:ODH-O2iM-7_WarmUp",
                                 "ConnLost" := "EPICS_PLC_Tester".#"HCB-TCH:ODH-O2iM-7_ConnLost",
                                 DEVICE_PARAM_OK=>#"HCB-TCH:ODH-O2iM-7");

      //********************************************
      // Device name: HCB-TCH:ODH-O2iM-8
      // Device type: ODH_O2iM
      //********************************************

      "DEV_HCB-TCH:ODH-O2iM-8_iDB" (
                                 "O2Level" := "EPICS_PLC_Tester".#"HCB-TCH:ODH-O2iM-8_O2Level",
                                 "ODHAlarm" := "EPICS_PLC_Tester".#"HCB-TCH:ODH-O2iM-8_ODHAlarm",
                                 "ODHWarning" := "EPICS_PLC_Tester".#"HCB-TCH:ODH-O2iM-8_ODHWarning",
                                 "MonitHealthy" := "EPICS_PLC_Tester".#"HCB-TCH:ODH-O2iM-8_MonitHealthy",
                                 "Maint" := "EPICS_PLC_Tester".#"HCB-TCH:ODH-O2iM-8_Maint",
                                 "MonitWarning" := "EPICS_PLC_Tester".#"HCB-TCH:ODH-O2iM-8_MonitWarning",
                                 "SysOK" := "EPICS_PLC_Tester".#"HCB-TCH:ODH-O2iM-8_SysOK",
                                 "WarmUp" := "EPICS_PLC_Tester".#"HCB-TCH:ODH-O2iM-8_WarmUp",
                                 "ConnLost" := "EPICS_PLC_Tester".#"HCB-TCH:ODH-O2iM-8_ConnLost",
                                 DEVICE_PARAM_OK=>#"HCB-TCH:ODH-O2iM-8");

      //********************************************
      // Device name: HCB-TCH:ODH-O2iM-9
      // Device type: ODH_O2iM
      //********************************************

      "DEV_HCB-TCH:ODH-O2iM-9_iDB" (
                                 "O2Level" := "EPICS_PLC_Tester".#"HCB-TCH:ODH-O2iM-9_O2Level",
                                 "ODHAlarm" := "EPICS_PLC_Tester".#"HCB-TCH:ODH-O2iM-9_ODHAlarm",
                                 "ODHWarning" := "EPICS_PLC_Tester".#"HCB-TCH:ODH-O2iM-9_ODHWarning",
                                 "MonitHealthy" := "EPICS_PLC_Tester".#"HCB-TCH:ODH-O2iM-9_MonitHealthy",
                                 "Maint" := "EPICS_PLC_Tester".#"HCB-TCH:ODH-O2iM-9_Maint",
                                 "MonitWarning" := "EPICS_PLC_Tester".#"HCB-TCH:ODH-O2iM-9_MonitWarning",
                                 "SysOK" := "EPICS_PLC_Tester".#"HCB-TCH:ODH-O2iM-9_SysOK",
                                 "WarmUp" := "EPICS_PLC_Tester".#"HCB-TCH:ODH-O2iM-9_WarmUp",
                                 "ConnLost" := "EPICS_PLC_Tester".#"HCB-TCH:ODH-O2iM-9_ConnLost",
                                 DEVICE_PARAM_OK=>#"HCB-TCH:ODH-O2iM-9");

      //********************************************
      // Device name: CXB-CXH:ODH-RIO-2
      // Device type: ODH_Rack
      //********************************************

      "DEV_CXB-CXH:ODH-RIO-2_iDB" (
                                 "SurgeArrOK" := "EPICS_PLC_Tester".#"CXB-CXH:ODH-RIO-2_SurgeArrOK",
                                 "PS24vOK" := "EPICS_PLC_Tester".#"CXB-CXH:ODH-RIO-2_PS24vOK",
                                 "UPSBatOK" := "EPICS_PLC_Tester".#"CXB-CXH:ODH-RIO-2_UPSBatOK",
                                 "UPS24vOK" := "EPICS_PLC_Tester".#"CXB-CXH:ODH-RIO-2_UPS24vOK",
                                 "UPSBuffReady" := "EPICS_PLC_Tester".#"CXB-CXH:ODH-RIO-2_UPSBuffReady",
                                 "UPSBatt85" := "EPICS_PLC_Tester".#"CXB-CXH:ODH-RIO-2_UPSBatt85",
                                 "UPSAlarm" := "EPICS_PLC_Tester".#"CXB-CXH:ODH-RIO-2_UPSAlarm",
                                 DEVICE_PARAM_OK=>#"CXB-CXH:ODH-RIO-2");

      //********************************************
      // Device name: HCB-ACH:ODH-RIO-1
      // Device type: ODH_Rack
      //********************************************

      "DEV_HCB-ACH:ODH-RIO-1_iDB" (
                                 "SurgeArrOK" := "EPICS_PLC_Tester".#"HCB-ACH:ODH-RIO-1_SurgeArrOK",
                                 "PS24vOK" := "EPICS_PLC_Tester".#"HCB-ACH:ODH-RIO-1_PS24vOK",
                                 "UPSBatOK" := "EPICS_PLC_Tester".#"HCB-ACH:ODH-RIO-1_UPSBatOK",
                                 "UPS24vOK" := "EPICS_PLC_Tester".#"HCB-ACH:ODH-RIO-1_UPS24vOK",
                                 "UPSBuffReady" := "EPICS_PLC_Tester".#"HCB-ACH:ODH-RIO-1_UPSBuffReady",
                                 "UPSBatt85" := "EPICS_PLC_Tester".#"HCB-ACH:ODH-RIO-1_UPSBatt85",
                                 "UPSAlarm" := "EPICS_PLC_Tester".#"HCB-ACH:ODH-RIO-1_UPSAlarm",
                                 DEVICE_PARAM_OK=>#"HCB-ACH:ODH-RIO-1");

      //********************************************
      // Device name: TS2-020Row:CnPw-U-001
      // Device type: ODH_Rack
      //********************************************

      "DEV_TS2-020Row:CnPw-U-001_iDB" (
                                 "SurgeArrOK" := "EPICS_PLC_Tester".#"TS2-020Row:CnPw-U-001_SurgeArrOK",
                                 "PS24vOK" := "EPICS_PLC_Tester".#"TS2-020Row:CnPw-U-001_PS24vOK",
                                 "UPSBatOK" := "EPICS_PLC_Tester".#"TS2-020Row:CnPw-U-001_UPSBatOK",
                                 "UPS24vOK" := "EPICS_PLC_Tester".#"TS2-020Row:CnPw-U-001_UPS24vOK",
                                 "UPSBuffReady" := "EPICS_PLC_Tester".#"TS2-020Row:CnPw-U-001_UPSBuffReady",
                                 "UPSBatt85" := "EPICS_PLC_Tester".#"TS2-020Row:CnPw-U-001_UPSBatt85",
                                 "UPSAlarm" := "EPICS_PLC_Tester".#"TS2-020Row:CnPw-U-001_UPSAlarm",
                                 DEVICE_PARAM_OK=>#"TS2-020Row:CnPw-U-001");
END_FUNCTION
TYPE "typeModul"
VERSION : 0.1
   STRUCT
      slotLaddr : HW_IO;   // Hardware ID of  module
      slotErrorState : Bool;   // error state of module
   END_STRUCT;

END_TYPE


TYPE "typeDevice"
VERSION : 0.1
   STRUCT
      laddr : HW_DEVICE;   // Logical address of a device or slave (system constant in HW configuration)
      "name" : String[50];   // Device name
      errorState : USInt;   // Status of the device 1=ok!, 2=faulty, 3=lost connection, 4=disabled, 12= was faulty, 13=was lost, 14=was disabled
      error : Bool;   // Signalizes an error in the device/slave
      nextDevice : Int;   // device number of next device
      actualConfiguredModules : Int;   // Actual number of configured modules in the device
      slot : Array[0..10] of "typeModul";   // slot informations
   END_STRUCT;

END_TYPE


TYPE "typeIoSystem"
VERSION : 0.1
   STRUCT
      ioSystemId : UInt;   // ID of  IO System
      ioSystemError : Bool;   // TRUE: if an error is occured in the assigned IO System
      firstDevice : Int := 0;   // device number (index) of first device in IO System
      lastDevice : Int := 0;   // device number (index) of last device IO System
      actualConfiguredDevices : Int := 0;   // Actual number of configured devices in the IO System
      device : Array[1..1] of "typeDevice";   // List of all devices in the IO System
   END_STRUCT;

END_TYPE

TYPE "typePlc"
VERSION : 0.1
   STRUCT
      actualConfiguredCentralModules : Int;   // Actual number of configured local modules
      errorState : Bool;   // Status of the device 1=ok!, 2=faulty, 3=lost connection, 4=disabled, 12= was faulty, 13=was lost, 14=was disabled
      slot : Array[1..10] of "typeModul";   // slot informations
   END_STRUCT;

END_TYPE



DATA_BLOCK "DiagnosticsData"
TITLE = Diagosis data DB
{ S7_Optimized_Access := 'TRUE' }
AUTHOR : SIEMENS
FAMILY : Diagnose
NAME : '10'
VERSION : 0.1
NON_RETAIN
//The global data block contains the data structure of the IO system, the control, the devices with the modules and an error buffer.
   VAR
      plc : "typePlc";   // diagnosis information PLC
      ioSystem : Array[1..5] of "typeIoSystem";   // diagnosis information IO systems
   END_VAR


BEGIN

END_DATA_BLOCK

FUNCTION_BLOCK "DiagStartupIoSystem"
{ S7_Optimized_Access := 'TRUE' }
VERSION : 0.1
   VAR_INPUT DB_SPECIFIC
      ioSystemHwId : HW_IOSYSTEM;   // This ID is representing the IO System (PN or DP), find the ID in the system constants
   END_VAR

   VAR_OUTPUT
      status : Int;   // The return value of system function, where the last error occured
      instructionError : Int;   // Indicates in which system function the error occured: 1= DeviceStates PN , 2=GetName PN, 3=ModuleStates PN,  4=DeviceStates DP, 5= GetName DP. 6= ModuleStates DP
      errorIndex : Int;   // The last index of the respective loop, if an error occures
   END_VAR

   VAR_IN_OUT
      ioSystem : "typeIoSystem";   // The diagnostics structure for one IO System
   END_VAR

   VAR
      statActualConfiguredDevices : Int := 0;   // Actual number of devices in the PN IO System
      statGeoAddr {OriginalPartName := 'GEOADDR'; LibVersion := '1.0'; ExternalAccessible := 'False'; ExternalVisible := 'False'; ExternalWritable := 'False'} : GEOADDR;   // Slot information
      statGeoLaddr { ExternalAccessible := 'False'; ExternalVisible := 'False'; ExternalWritable := 'False'} : HW_ANY;   // GEO2LOG hardware identifier
      statConfiguredDevices { ExternalAccessible := 'False'; ExternalVisible := 'False'; ExternalWritable := 'False'} : Array[0..1023] of Bool;   // Temporary storage of the return of "DeviceStates", to combine the states of the devices with numbers and names
      statExistingDevices : Array[0..1023] of Bool;   // Temporary storage of the return of "DeviceStates", to combine the states of the devices with numbers and names
      statFaultyDevices : Array[0..1023] of Bool;   // Temporary storage of the return of "DeviceStates", to combine the states of the divices with numbers and names
      statDisabledDevices { ExternalAccessible := 'False'; ExternalVisible := 'False'; ExternalWritable := 'False'} : Array[0..1023] of Bool;   // Storage of the status of all devices in the PN IO System --> State: Disabled
      statProblemDevices { ExternalAccessible := 'False'; ExternalVisible := 'False'; ExternalWritable := 'False'} : Array[0..1023] of Bool;   // Storage of the status of all devices in the PN IO System --> State: Problem
      statDeviceModuleStates : Array[0..127] of Bool;   // Storage of the status of all modules in the PN Devices --> State: Problem
      instGetNameDevices {OriginalPartName := 'FB_806_S71500'; LibVersion := '1.3'} : Get_Name;   // Instance of system function "GetName"
      statInitString : String;   // Used to initialize the temporary string to convert into STRING[50]
      statFirstDevice : UInt;   // Station number of the first device of the list
      statFirstDeviceFlag { ExternalAccessible := 'False'; ExternalVisible := 'False'; ExternalWritable := 'False'} : Bool := TRUE;   // Help tag for the first device in the linked list
      statLastDevice : UInt;   // Station number of the last device of the list
      statLinkedListPointer : Int;   // The actual index pointer of the linked list (Actual pointer = Station number of the device)
      statFirstRun : Bool := TRUE;   // Signalizes the first run
      statResetStatesOld : Bool;   // Detect a rising edge at ResetStates
      statMaxDevices : Int;
   END_VAR

   VAR_TEMP
      tempIndex : Int;   // index configured devices
      tempSlotIndex : Int;   // Loop index
      tempModuleNum : Int;   // index module number
      tempRetValGeo : Int;   // GEO2LOG error information
      tempRetValDeviceStates : Int;   // DeviceStates error information
      tempRetValModuleStates : Int;   // Return value system function ModuleStates
      tempStringConvert : String;   // Store the device names temporary here, to convert them into STRING[50]
      tempLastDevice : UInt;   // Temporary storage of the actual index, if it is the last device --> store it in static
      tempIoSystemError : Bool;
   END_VAR

   VAR CONSTANT
      STATE_CONFIGURED : USInt := 1;   // Used for instruction DeviceStates, read out all configured devices
      STATE_FAULTY : USInt := 2;   // Used for instruction DeviceStates, read out all faulty devices
      STATE_DISABLED : USInt := 3;   // Used for instruction DeviceStates, read out all disabled devices
      STATE_EXIST : USInt := 4;   // Used for instruction DeviceStates, read out all devices not reachable
      STATE_PROBLEM : USInt := 5;   // Used for instruction DeviceStates, read out all devices with several problems
      DEVICE_SLAVE : USInt := 2;   // GEO2LOG structure: HW type = 2
      MODULE_OF_DEVICE : USInt := 4;   // GEO2LOG structure: HW type = 4
      IO_SYSTEM_AREA : USInt := 1;   // GEO2LOG structure: Area = 1
      DP_SYSTEM_AREA : USInt := 2;   // GEO2LOG structure: Area = 2
      ERR_DEV_STATE_DEVICES : USInt := 1;   // Identifies the instruction behind the error code of output "Status" --> DeviceStates PN (Configured, faulty, existing)
      ERR_GET_NAME_DEVICES : USInt := 2;   // Identifies the instruction behind the error code of output "Status" -->  GetName of devices PN
      ERR_MOD_STAT_DEVICES : USInt := 3;   // Identifies the instruction behind the error code of output "Status" --> ModuleStates PN
      ERR_DEV_STAT_PN : USInt := 1;   // Value for output instruction error, DeviceStates PN devices
      ERR_MOD_STAT_PN : USInt := 4;   // Value for output instruction error, ModuleStates PN devices
      MAX_SLAVES_DP : Int := 127;
      MAX_SLAVES_PN : Int := 127;
   END_VAR


BEGIN
	//=============================================================================
	//Author: SIEMENS, Owner: Miklos Boros
	//        email: borosmiklos@gmail.com; miklos.boros@esss.se
	//
	//Functionality: Determine hardware identifier and module states from
	//               PN or DP IO system
	//
	//
	//Please Note:
	//        This block is part of the generated ESS Standard Code
	//        DON'T CHANGE THIS BLOCK MANUALY. Any changes will be overwritten in the next code generation.
	//
	//
	//Change log table:
	//Version  Date         Expert in charge      Changes applied
	//01.00.00 29.08.2017   ESS/ICS               First released version for PLCFactory
	//02.00.00 09-04-2018   ESS/ICS               Major bug fix for PN/DP devices
	//=============================================================================


	// The startup will be executed only once --> initialize the first run
	// indicator.
	#statFirstDeviceFlag := TRUE;
	#statFirstRun := TRUE;
	#statActualConfiguredDevices := 0;
	#statFirstDevice := 1;
	#statLastDevice := 1;

	//=============================================================================
	// CONFIGURED DEVICES
	//=============================================================================
	// Find out how much devices are configured in the IO System --> PROFINET IO
	// This number is the maximum number of devices, which will be checked in the
	// following programm
	#tempRetValDeviceStates := DeviceStates(LADDR := #ioSystemHwId,
	                                        MODE := #STATE_CONFIGURED,
	                                        STATE := #statConfiguredDevices);

	// Check if the block call was successful
	IF (#tempRetValDeviceStates <> 0)
	THEN
	    // Error handling
	    #status := #tempRetValDeviceStates;
	    #instructionError := #ERR_DEV_STATE_DEVICES;
	    // Call ok --> store the actual number of configured devices
	ELSE
	    ;
	END_IF;

